C01815=1039.477,-0.924,417.452,169.236,37.751,157.096
C01816=1039.483,-0.675,417.437,169.238,37.752,157.096
C01817=1039.489,-0.426,417.422,169.240,37.752,157.096
C01818=1039.495,-0.176,417.407,169.242,37.753,157.096
C01819=1039.502,0.074,417.392,169.244,37.754,157.096
C01820=1039.508,0.323,417.378,169.246,37.754,157.096
C01821=1039.515,0.572,417.362,169.248,37.754,157.097
C01822=1039.520,0.822,417.347,169.250,37.755,157.097
C01823=1039.526,1.071,417.332,169.253,37.755,157.097
C01824=1039.533,1.321,417.317,169.255,37.756,157.097
C01825=1039.539,1.571,417.302,169.257,37.756,157.097
C01826=1039.545,1.820,417.287,169.259,37.757,157.097
C01827=1039.551,2.069,417.272,169.262,37.758,157.097
C01828=1039.558,2.319,417.257,169.264,37.758,157.098
C01829=1039.564,2.568,417.242,169.266,37.759,157.098
C01830=1039.571,2.817,417.227,169.268,37.759,157.098
C01831=1039.577,3.067,417.212,169.270,37.760,157.098
C01832=1039.583,3.317,417.197,169.272,37.760,157.098
C01833=1039.589,3.566,417.182,169.275,37.761,157.098
C01834=1039.596,3.815,417.167,169.277,37.762,157.098
C01835=1039.602,4.065,417.152,169.279,37.762,157.099
C01836=1039.609,4.314,417.137,169.281,37.763,157.099
C01837=1039.615,4.564,417.122,169.283,37.763,157.099
C01838=1039.621,4.813,417.107,169.285,37.763,157.099
C01839=1039.627,5.063,417.091,169.287,37.764,157.099
C01840=1039.634,5.313,417.076,169.289,37.764,157.099
C01841=1039.640,5.561,417.061,169.291,37.765,157.099
C01842=1039.646,5.811,417.046,169.293,37.766,157.099
C01843=1039.652,6.061,417.031,169.296,37.766,157.099
C01844=1039.659,6.310,417.016,169.298,37.767,157.100
C01845=1039.665,6.559,417.001,169.300,37.767,157.100
C01846=1039.672,6.809,416.986,169.302,37.768,157.100
C01847=1039.678,7.059,416.971,169.304,37.768,157.100
C01848=1039.685,7.308,416.956,169.306,37.769,157.100
C01849=1039.691,7.557,416.940,169.308,37.770,157.100
C01850=1039.698,7.807,416.925,169.310,37.770,157.100
C01851=1039.703,8.057,416.910,169.312,37.770,157.100
C01852=1039.710,8.306,416.894,169.314,37.771,157.101
C01853=1039.716,8.556,416.879,169.316,37.771,157.101
C01854=1039.723,8.805,416.864,169.319,37.772,157.101
C01855=1039.729,9.054,416.849,169.321,37.772,157.101
C01856=1039.735,9.303,416.834,169.322,37.773,157.101
C01857=1039.742,9.553,416.819,169.324,37.774,157.101
C01858=1039.748,9.802,416.803,169.326,37.774,157.101
C01859=1039.755,10.052,416.788,169.328,37.775,157.102
C01860=1039.761,10.301,416.773,169.330,37.775,157.102
C01861=1039.767,10.551,416.757,169.332,37.776,157.102
C01862=1039.773,10.800,416.742,169.334,37.776,157.102
C01863=1039.780,11.049,416.726,169.336,37.777,157.102
C01864=1039.786,11.299,416.711,169.338,37.777,157.102
C01865=1039.793,11.549,416.697,169.341,37.778,157.102
C01866=1039.800,11.798,416.681,169.343,37.778,157.102
C01867=1039.806,12.047,416.666,169.345,37.779,157.102
C01868=1039.813,12.333,416.648,169.348,37.779,157.103
C01869=1039.821,12.618,416.631,169.350,37.780,157.103
C01870=1039.827,12.904,416.613,169.352,37.780,157.103
C01871=1039.835,13.189,416.595,169.354,37.781,157.103
C01872=1039.842,13.438,416.580,169.356,37.782,157.103
C01873=1039.848,13.688,416.565,169.358,37.782,157.103
C01874=1039.855,13.938,416.549,169.361,37.783,157.103
C01875=1039.862,14.187,416.534,169.363,37.783,157.104
C01876=1039.868,14.437,416.517,169.365,37.784,157.104
C01877=1039.874,14.686,416.503,169.367,37.784,157.104
C01878=1039.881,14.935,416.487,169.369,37.785,157.104
C01879=1039.886,15.185,416.471,169.371,37.786,157.104
C01880=1039.893,15.434,416.456,169.373,37.786,157.104
C01881=1039.900,15.683,416.440,169.375,37.787,157.104
C01882=1039.905,15.933,416.424,169.377,37.787,157.105
C01883=1039.912,16.182,416.409,169.379,37.788,157.105
C01884=1039.918,16.432,416.393,169.382,37.788,157.105
C01885=1039.924,16.681,416.378,169.384,37.789,157.105
C01886=1039.931,16.930,416.362,169.386,37.790,157.105
C01887=1039.937,17.180,416.346,169.388,37.791,157.105
C01888=1039.944,17.429,416.331,169.390,37.791,157.105
C01889=1039.949,17.679,416.314,169.392,37.792,157.106
C01890=1039.956,17.928,416.300,169.393,37.793,157.106
C01891=1039.963,18.177,416.284,169.395,37.793,157.106
C01892=1039.968,18.427,416.268,169.397,37.794,157.106
C01893=1039.975,18.677,416.252,169.400,37.794,157.106
C01894=1039.982,18.926,416.237,169.402,37.795,157.106
C01895=1039.988,19.176,416.220,169.404,37.795,157.106
C01896=1039.994,19.425,416.205,169.406,37.796,157.107
C01897=1040.000,19.675,416.189,169.408,37.797,157.107
C01898=1040.007,19.924,416.174,169.410,37.797,157.107
C01899=1040.013,20.174,416.158,169.412,37.798,157.107
C01900=1040.019,20.423,416.142,169.414,37.798,157.107
C01901=1040.025,20.672,416.126,169.416,37.799,157.107
C01902=1040.032,20.921,416.110,169.419,37.799,157.107
C01903=1040.039,21.171,416.094,169.420,37.800,157.107
C01904=1040.045,21.421,416.079,169.422,37.801,157.108
C01905=1040.051,21.670,416.063,169.424,37.802,157.108
C01906=1040.058,21.919,416.047,169.426,37.802,157.108
C01907=1040.064,22.168,416.031,169.428,37.803,157.108
C01908=1040.070,22.417,416.015,169.430,37.804,157.108
C01909=1040.076,22.667,415.999,169.432,37.804,157.108
C01910=1040.083,22.917,415.983,169.434,37.805,157.109
C01911=1040.089,23.167,415.967,169.437,37.805,157.109
C01912=1040.095,23.416,415.951,169.439,37.806,157.109
C01913=1040.102,23.665,415.935,169.441,37.806,157.109
C01914=1040.108,23.914,415.919,169.442,37.808,157.109
C01915=1040.114,24.164,415.904,169.444,37.808,157.109
C01916=1040.120,24.413,415.888,169.446,37.809,157.109
C01917=1040.127,24.663,415.872,169.448,37.809,157.110
C01918=1040.133,24.912,415.855,169.450,37.810,157.110
C01919=1040.140,25.161,415.840,169.452,37.811,157.110
C01920=1040.146,25.411,415.824,169.455,37.811,157.110
C01921=1040.152,25.660,415.807,169.457,37.812,157.110
C01922=1040.159,25.910,415.791,169.459,37.812,157.110
C01923=1040.165,26.159,415.775,169.461,37.813,157.110
C01924=1040.172,26.408,415.759,169.463,37.813,157.111
C01925=1040.178,26.658,415.743,169.464,37.814,157.111
C01926=1040.185,26.907,415.727,169.466,37.815,157.111
C01927=1040.191,27.157,415.711,169.468,37.816,157.111
C01928=1040.197,27.407,415.695,169.470,37.816,157.111
C01929=1040.203,27.656,415.680,169.473,37.817,157.111
C01930=1040.209,27.905,415.663,169.475,37.817,157.111
C01931=1040.216,28.155,415.647,169.477,37.818,157.112
C01932=1040.223,28.441,415.628,169.479,37.819,157.112
C01933=1040.231,28.728,415.609,169.481,37.820,157.112
C01934=1040.238,29.014,415.592,169.483,37.820,157.112
C01935=1040.244,29.301,415.572,169.485,37.821,157.112
C01936=1040.252,29.551,415.556,169.488,37.822,157.113
C01937=1040.258,29.800,415.540,169.490,37.823,157.113
C01938=1040.264,30.049,415.524,169.492,37.823,157.113
C01939=1040.270,30.299,415.508,169.494,37.824,157.113
C01940=1040.276,30.548,415.490,169.496,37.824,157.113
C01941=1040.283,30.797,415.475,169.498,37.826,157.113
C01942=1040.289,31.047,415.458,169.500,37.826,157.113
C01943=1040.295,31.296,415.442,169.501,37.827,157.114
C01944=1040.302,31.546,415.425,169.503,37.827,157.114
C01945=1040.308,31.795,415.410,169.506,37.828,157.114
C01946=1040.314,32.044,415.393,169.508,37.829,157.114
C01947=1040.321,32.293,415.376,169.510,37.830,157.114
C01948=1040.327,32.543,415.360,169.512,37.830,157.114
C01949=1040.333,32.793,415.344,169.514,37.831,157.115
C01950=1040.340,33.042,415.328,169.515,37.832,157.115
C01951=1040.346,33.292,415.311,169.517,37.832,157.115
C01952=1040.352,33.541,415.295,169.519,37.833,157.115
C01953=1040.358,33.790,415.278,169.522,37.834,157.115
C01954=1040.365,34.040,415.261,169.524,37.834,157.115
C01955=1040.372,34.289,415.246,169.526,37.835,157.115
C01956=1040.378,34.538,415.230,169.528,37.836,157.116
C01957=1040.384,34.788,415.213,169.530,37.836,157.116
C01958=1040.390,35.037,415.196,169.531,37.837,157.116
C01959=1040.396,35.286,415.180,169.533,37.838,157.116
C01960=1040.403,35.536,415.163,169.535,37.839,157.116
C01961=1040.410,35.785,415.147,169.537,37.839,157.116
C01962=1040.416,36.034,415.130,169.540,37.840,157.117
C01963=1040.422,36.284,415.114,169.542,37.840,157.117
C01964=1040.428,36.533,415.098,169.544,37.841,157.117
C01965=1040.435,36.782,415.081,169.546,37.841,157.117
C01966=1040.442,37.032,415.065,169.547,37.843,157.117
C01967=1040.448,37.281,415.048,169.549,37.843,157.117
C01968=1040.454,37.531,415.032,169.551,37.844,157.117
C01969=1040.461,37.780,415.015,169.553,37.844,157.118
C01970=1040.467,38.029,414.998,169.556,37.845,157.118
C01971=1040.473,38.278,414.981,169.558,37.846,157.118
C01972=1040.479,38.528,414.965,169.559,37.847,157.118
C01973=1040.485,38.778,414.949,169.561,37.847,157.118
C01974=1040.492,39.027,414.931,169.563,37.848,157.119
C01975=1040.498,39.276,414.915,169.565,37.849,157.119
C01976=1040.505,39.525,414.898,169.567,37.850,157.119
C01977=1040.510,39.775,414.881,169.569,37.850,157.119
C01978=1040.516,40.025,414.865,169.571,37.851,157.119
C01979=1040.523,40.273,414.848,169.573,37.852,157.119
C01980=1040.529,40.524,414.831,169.575,37.853,157.119
C01981=1040.535,40.772,414.814,169.577,37.853,157.120
C01982=1040.542,41.022,414.797,169.579,37.854,157.120
C01983=1040.548,41.271,414.780,169.581,37.855,157.120
C01984=1040.554,41.520,414.764,169.582,37.855,157.120
C01985=1040.561,41.770,414.747,169.584,37.856,157.120
C01986=1040.567,42.019,414.731,169.587,37.857,157.121
C01987=1040.574,42.269,414.713,169.589,37.858,157.121
C01988=1040.580,42.518,414.697,169.591,37.858,157.121
C01989=1040.586,42.767,414.680,169.593,37.859,157.121
C01990=1040.593,43.017,414.663,169.594,37.860,157.121
C01991=1040.599,43.265,414.646,169.596,37.861,157.121
C01992=1040.605,43.516,414.629,169.598,37.861,157.121
C01993=1040.611,43.765,414.612,169.601,37.862,157.122
C01994=1040.617,44.015,414.596,169.603,37.863,157.122
C01995=1040.624,44.263,414.579,169.605,37.864,157.122
C01996=1040.630,44.550,414.559,169.607,37.865,157.122
C01997=1040.638,44.837,414.539,169.609,37.865,157.122
C01998=1040.645,45.123,414.520,169.611,37.867,157.123
C01999=1040.652,45.410,414.500,169.614,37.868,157.123
C02000=1040.658,45.659,414.483,169.616,37.868,157.123
C02001=1040.664,45.908,414.466,169.617,37.869,157.123
C02002=1040.670,46.158,414.449,169.619,37.870,157.123
C02003=1040.676,46.407,414.432,169.621,37.871,157.124
C02004=1040.682,46.657,414.414,169.623,37.871,157.124
C02005=1040.688,46.906,414.398,169.625,37.873,157.124
C02006=1040.695,47.155,414.381,169.626,37.873,157.124
C02007=1040.701,47.404,414.363,169.629,37.874,157.124
C02008=1040.707,47.654,414.347,169.631,37.875,157.125
C02009=1040.714,47.903,414.329,169.633,37.875,157.125
C02010=1040.720,48.152,414.312,169.635,37.876,157.125
C02011=1040.726,48.402,414.294,169.636,37.877,157.125
C02012=1040.732,48.651,414.278,169.638,37.878,157.125
C02013=1040.739,48.900,414.261,169.640,37.879,157.125
C02014=1040.744,49.150,414.243,169.643,37.880,157.126
C02015=1040.751,49.399,414.226,169.645,37.880,157.126
C02016=1040.757,49.648,414.210,169.646,37.881,157.126
C02017=1040.763,49.898,414.192,169.648,37.882,157.126
C02018=1040.770,50.147,414.175,169.650,37.883,157.126
C02019=1040.776,50.396,414.157,169.652,37.884,157.126
C02020=1040.782,50.645,414.140,169.654,37.884,157.127
C02021=1040.788,50.895,414.123,169.656,37.885,157.127
C02022=1040.795,51.144,414.106,169.658,37.886,157.127
C02023=1040.801,51.394,414.088,169.660,37.887,157.127
C02024=1040.809,51.733,414.065,169.663,37.888,157.127
C02025=1040.818,52.073,414.041,169.665,37.888,157.128
C02026=1040.827,52.412,414.018,169.667,37.890,157.128
C02027=1040.835,52.751,413.995,169.671,37.891,157.128
C02028=1040.841,53.001,413.977,169.673,37.891,157.128
C02029=1040.847,53.250,413.960,169.675,37.893,157.128
C02030=1040.854,53.500,413.943,169.676,37.893,157.129
C02031=1040.860,53.749,413.925,169.678,37.894,157.129
C02032=1040.866,53.998,413.908,169.680,37.895,157.129
C02033=1040.873,54.247,413.891,169.682,37.895,157.129
C02034=1040.879,54.497,413.873,169.685,37.896,157.129
C02035=1040.886,54.746,413.856,169.686,37.897,157.130
C02036=1040.893,54.995,413.839,169.688,37.898,157.130
C02037=1040.898,55.244,413.821,169.690,37.898,157.130
C02038=1040.905,55.494,413.804,169.692,37.899,157.130
C02039=1040.910,55.743,413.787,169.694,37.900,157.130
C02040=1040.917,55.993,413.769,169.695,37.901,157.130
C02041=1040.924,56.242,413.752,169.697,37.901,157.130
C02042=1040.929,56.491,413.735,169.700,37.903,157.131
C02043=1040.936,56.741,413.717,169.702,37.903,157.131
C02044=1040.943,56.990,413.700,169.704,37.904,157.131
C02045=1040.949,57.239,413.682,169.705,37.904,157.131
C02046=1040.955,57.489,413.665,169.707,37.905,157.131
C02047=1040.961,57.738,413.647,169.709,37.906,157.132
C02048=1040.968,57.987,413.630,169.711,37.907,157.132
C02049=1040.975,58.237,413.613,169.714,37.908,157.132
C02050=1040.980,58.486,413.595,169.715,37.908,157.132
C02051=1040.987,58.735,413.578,169.717,37.909,157.132
C02052=1040.993,58.985,413.560,169.719,37.910,157.132
C02053=1041.000,59.234,413.543,169.721,37.911,157.133
C02054=1041.006,59.483,413.526,169.723,37.911,157.133
C02055=1041.013,59.732,413.507,169.725,37.912,157.133
C02056=1041.019,59.955,413.492,169.726,37.912,157.133
C02057=1041.024,60.178,413.476,169.729,37.913,157.133
C02058=1041.030,60.401,413.461,169.730,37.914,157.133
C02059=1041.036,60.623,413.445,169.732,37.915,157.134
C02060=1041.041,60.845,413.429,169.734,37.915,157.134
C02061=1041.047,61.068,413.413,169.735,37.916,157.134
C02062=1041.053,61.292,413.398,169.737,37.917,157.134
C02063=1041.058,61.514,413.382,169.739,37.917,157.134
C02064=1041.065,61.763,413.365,169.740,37.918,157.134
C02065=1041.071,62.013,413.347,169.743,37.919,157.134
C02066=1041.078,62.262,413.329,169.745,37.919,157.135
C02067=1041.084,62.511,413.312,169.747,37.920,157.135
C02068=1041.091,62.760,413.294,169.749,37.921,157.135
C02069=1041.097,63.010,413.276,169.750,37.922,157.135
C02070=1041.104,63.259,413.259,169.752,37.922,157.135
C02071=1041.110,63.508,413.242,169.754,37.923,157.135
C02072=1041.116,63.757,413.223,169.756,37.923,157.136
C02073=1041.123,64.007,413.206,169.759,37.925,157.136
C02074=1041.129,64.257,413.188,169.760,37.925,157.136
C02075=1041.135,64.506,413.171,169.762,37.926,157.136
C02076=1041.142,64.755,413.153,169.764,37.927,157.136
C02077=1041.148,65.004,413.135,169.766,37.928,157.136
C02078=1041.154,65.254,413.117,169.768,37.929,157.137
C02079=1041.160,65.503,413.100,169.769,37.929,157.137
C02080=1041.167,65.752,413.081,169.772,37.930,157.137
C02081=1041.173,66.001,413.063,169.774,37.931,157.137
C02082=1041.179,66.251,413.045,169.776,37.932,157.137
C02083=1041.185,66.500,413.028,169.778,37.933,157.138
C02084=1041.192,66.749,413.010,169.779,37.933,157.138
C02085=1041.198,66.999,412.992,169.781,37.934,157.138
C02086=1041.205,67.248,412.974,169.783,37.935,157.138
C02087=1041.211,67.497,412.956,169.786,37.936,157.138
C02088=1041.217,67.746,412.938,169.787,37.936,157.138
C02089=1041.223,67.995,412.919,169.789,37.938,157.139
C02090=1041.230,68.245,412.902,169.791,37.938,157.139
C02091=1041.236,68.495,412.884,169.793,37.939,157.139
C02092=1041.242,68.743,412.866,169.795,37.940,157.139
C02093=1041.248,68.993,412.848,169.796,37.940,157.139
C02094=1041.255,69.242,412.831,169.799,37.942,157.140
C02095=1041.261,69.491,412.812,169.801,37.942,157.140
C02096=1041.267,69.740,412.794,169.803,37.943,157.140
C02097=1041.273,69.990,412.776,169.804,37.944,157.140
C02098=1041.279,70.239,412.758,169.806,37.945,157.140
C02099=1041.286,70.488,412.739,169.808,37.946,157.141
C02100=1041.293,70.738,412.722,169.810,37.946,157.141
C02101=1041.299,70.986,412.703,169.813,37.948,157.141
C02102=1041.305,71.236,412.686,169.814,37.948,157.141
C02103=1041.311,71.485,412.667,169.816,37.949,157.141
C02104=1041.317,71.735,412.649,169.818,37.950,157.142
C02105=1041.324,71.984,412.630,169.820,37.951,157.142
C02106=1041.329,72.233,412.613,169.821,37.952,157.142
C02107=1041.336,72.482,412.594,169.824,37.953,157.142
C02108=1041.342,72.732,412.576,169.826,37.953,157.142
C02109=1041.349,72.981,412.558,169.828,37.954,157.142
C02110=1041.355,73.230,412.540,169.830,37.955,157.143
C02111=1041.361,73.480,412.522,169.831,37.956,157.143
C02112=1041.367,73.729,412.504,169.833,37.957,157.143
C02113=1041.373,73.978,412.485,169.835,37.958,157.143
C02114=1041.380,74.227,412.467,169.838,37.959,157.144
C02115=1041.386,74.477,412.449,169.839,37.959,157.144
C02116=1041.392,74.726,412.430,169.841,37.960,157.144
C02117=1041.398,74.975,412.412,169.843,37.961,157.144
C02118=1041.405,75.225,412.394,169.845,37.962,157.144
C02119=1041.411,75.473,412.375,169.847,37.963,157.144
C02120=1041.417,75.723,412.357,169.849,37.963,157.145
C02121=1041.423,75.972,412.339,169.851,37.965,157.145
C02122=1041.430,76.221,412.321,169.853,37.965,157.145
C02123=1041.437,76.470,412.303,169.855,37.966,157.145
C02124=1041.444,76.757,412.281,169.857,37.967,157.145
C02125=1041.451,77.042,412.260,169.859,37.968,157.146
C02126=1041.458,77.329,412.239,169.861,37.969,157.146
C02127=1041.465,77.615,412.218,169.864,37.970,157.146
C02128=1041.471,77.864,412.199,169.866,37.970,157.146
C02129=1041.477,78.113,412.181,169.867,37.972,157.146
C02130=1041.483,78.363,412.163,169.869,37.972,157.147
C02131=1041.490,78.612,412.144,169.871,37.973,157.147
C02132=1041.496,78.861,412.126,169.873,37.974,157.147
C02133=1041.503,79.110,412.107,169.875,37.975,157.147
C02134=1041.509,79.360,412.089,169.877,37.976,157.148
C02135=1041.514,79.609,412.070,169.879,37.977,157.148
C02136=1041.521,79.858,412.051,169.881,37.978,157.148
C02137=1041.527,80.107,412.033,169.882,37.979,157.148
C02138=1041.533,80.356,412.014,169.884,37.980,157.148
C02139=1041.539,80.605,411.996,169.887,37.980,157.148
C02140=1041.545,80.855,411.977,169.889,37.982,157.149
C02141=1041.551,81.104,411.958,169.891,37.982,157.149
C02142=1041.558,81.353,411.940,169.892,37.983,157.149
C02143=1041.564,81.602,411.921,169.894,37.984,157.149
C02144=1041.571,81.851,411.902,169.896,37.985,157.150
C02145=1041.576,82.101,411.883,169.899,37.986,157.150
C02146=1041.582,82.351,411.865,169.900,37.987,157.150
C02147=1041.589,82.600,411.847,169.902,37.987,157.150
C02148=1041.595,82.849,411.828,169.904,37.989,157.150
C02149=1041.602,83.098,411.809,169.906,37.989,157.150
C02150=1041.607,83.347,411.790,169.907,37.990,157.151
C02151=1041.614,83.597,411.771,169.909,37.991,157.151
C02152=1041.620,83.846,411.753,169.912,37.992,157.151
C02153=1041.627,84.095,411.734,169.914,37.993,157.151
C02154=1041.633,84.344,411.716,169.916,37.994,157.152
C02155=1041.639,84.593,411.696,169.917,37.994,157.152
C02156=1041.645,84.842,411.678,169.919,37.996,157.152
C02157=1041.652,85.092,411.659,169.921,37.996,157.152
C02158=1041.658,85.341,411.641,169.924,37.997,157.152
C02159=1041.664,85.590,411.622,169.925,37.998,157.152
C02160=1041.670,85.840,411.603,169.927,37.999,157.153
C02161=1041.676,86.089,411.585,169.929,38.000,157.153
C02162=1041.683,86.338,411.566,169.931,38.001,157.153
C02163=1041.689,86.587,411.547,169.933,38.001,157.153
C02164=1041.695,86.837,411.528,169.935,38.003,157.153
C02165=1041.701,87.086,411.509,169.937,38.003,157.154
C02166=1041.708,87.335,411.491,169.939,38.004,157.154
C02167=1041.714,87.584,411.472,169.941,38.005,157.154
C02168=1041.720,87.833,411.453,169.942,38.006,157.154
C02169=1041.726,88.083,411.434,169.944,38.007,157.154
C02170=1041.733,88.331,411.415,169.947,38.008,157.155
C02171=1041.739,88.580,411.396,169.949,38.009,157.155
C02172=1041.746,88.829,411.377,169.951,38.010,157.155
C02173=1041.751,89.079,411.358,169.952,38.010,157.155
C02174=1041.758,89.328,411.340,169.954,38.011,157.155
C02175=1041.764,89.577,411.321,169.956,38.012,157.156
C02176=1041.771,89.826,411.302,169.958,38.013,157.156
C02177=1041.777,90.076,411.283,169.961,38.014,157.156
C02178=1041.783,90.325,411.264,169.962,38.014,157.156
C02179=1041.789,90.575,411.245,169.964,38.016,157.156
C02180=1041.796,90.823,411.225,169.966,38.017,157.157
C02181=1041.802,91.073,411.206,169.968,38.017,157.157
C02182=1041.808,91.322,411.188,169.969,38.019,157.157
C02183=1041.814,91.571,411.168,169.972,38.019,157.157
C02184=1041.820,91.820,411.150,169.974,38.020,157.157
C02185=1041.826,92.069,411.130,169.976,38.021,157.158
C02186=1041.833,92.318,411.111,169.977,38.022,157.158
C02187=1041.838,92.568,411.092,169.979,38.023,157.158
C02188=1041.845,92.854,411.070,169.982,38.024,157.158
C02189=1041.853,93.140,411.048,169.984,38.025,157.159
C02190=1041.860,93.426,411.026,169.986,38.026,157.159
C02191=1041.867,93.712,411.004,169.988,38.027,157.159
C02192=1041.873,93.961,410.985,169.990,38.028,157.159
C02193=1041.879,94.210,410.966,169.992,38.029,157.159
C02194=1041.885,94.459,410.946,169.995,38.030,157.160
C02195=1041.892,94.708,410.927,169.996,38.031,157.160
C02196=1041.898,94.958,410.908,169.998,38.032,157.160
C02197=1041.904,95.206,410.889,170.000,38.033,157.160
C02198=1041.911,95.456,410.869,170.002,38.034,157.161
C02199=1041.917,95.706,410.850,170.004,38.035,157.161
C02200=1041.923,95.955,410.831,170.006,38.036,157.161
C02201=1041.929,96.204,410.811,170.008,38.037,157.161
C02202=1041.935,96.453,410.793,170.010,38.037,157.161
C02203=1041.941,96.702,410.773,170.012,38.038,157.162
C02204=1041.948,96.951,410.754,170.014,38.039,157.162
C02205=1041.954,97.201,410.734,170.015,38.040,157.162
C02206=1041.961,97.449,410.715,170.018,38.041,157.162
C02207=1041.966,97.699,410.696,170.020,38.042,157.162
C02208=1041.973,97.948,410.677,170.022,38.043,157.163
C02209=1041.979,98.197,410.657,170.024,38.044,157.163
C02210=1041.985,98.446,410.639,170.025,38.045,157.163
C02211=1041.992,98.695,410.618,170.027,38.045,157.163
C02212=1041.997,98.945,410.599,170.030,38.047,157.163
C02213=1042.004,99.194,410.580,170.032,38.047,157.164
C02214=1042.010,99.443,410.560,170.034,38.048,157.164
C02215=1042.016,99.692,410.542,170.035,38.049,157.164
C02216=1042.023,99.941,410.521,170.037,38.050,157.164
C02217=1042.029,100.191,410.503,170.039,38.051,157.165
C02218=1042.035,100.439,410.483,170.042,38.052,157.165
C02219=1042.041,100.689,410.464,170.044,38.053,157.165
C02220=1042.048,100.937,410.444,170.045,38.054,157.165
C02221=1042.054,101.188,410.425,170.047,38.055,157.165
C02222=1042.060,101.436,410.405,170.049,38.056,157.166
C02223=1042.066,101.686,410.385,170.051,38.056,157.166
C02224=1042.072,101.935,410.365,170.053,38.058,157.166
C02225=1042.078,102.183,410.345,170.055,38.059,157.166
C02226=1042.085,102.433,410.326,170.057,38.059,157.166
C02227=1042.091,102.682,410.306,170.059,38.061,157.167
C02228=1042.096,102.931,410.287,170.061,38.062,157.167
C02229=1042.102,103.180,410.267,170.062,38.062,157.167
C02230=1042.108,103.429,410.247,170.065,38.064,157.167
C02231=1042.115,103.679,410.228,170.067,38.065,157.168
C02232=1042.121,103.928,410.208,170.069,38.065,157.168
C02233=1042.127,104.177,410.189,170.070,38.067,157.168
C02234=1042.133,104.426,410.169,170.072,38.068,157.168
C02235=1042.140,104.675,410.149,170.075,38.068,157.168
C02236=1042.146,104.925,410.130,170.077,38.069,157.169
C02237=1042.152,105.173,410.110,170.079,38.071,157.169
C02238=1042.158,105.422,410.090,170.080,38.071,157.169
C02239=1042.164,105.672,410.071,170.082,38.072,157.169
C02240=1042.170,105.921,410.051,170.085,38.074,157.170
C02241=1042.176,106.170,410.031,170.087,38.074,157.170
C02242=1042.183,106.419,410.012,170.089,38.075,157.170
C02243=1042.189,106.669,409.992,170.090,38.076,157.170
C02244=1042.195,106.917,409.972,170.092,38.077,157.170
C02245=1042.201,107.166,409.952,170.094,38.078,157.171
C02246=1042.208,107.416,409.932,170.096,38.079,157.171
C02247=1042.214,107.665,409.912,170.099,38.080,157.171
C02248=1042.220,107.914,409.893,170.100,38.081,157.171
C02249=1042.227,108.163,409.873,170.102,38.082,157.172
C02250=1042.233,108.413,409.853,170.104,38.083,157.172
C02251=1042.239,108.661,409.833,170.106,38.084,157.172
C02252=1042.245,108.947,409.810,170.109,38.085,157.172
C02253=1042.253,109.234,409.788,170.111,38.086,157.172
C02254=1042.260,109.520,409.765,170.113,38.087,157.173
C02255=1042.267,109.806,409.742,170.115,38.088,157.173
C02256=1042.273,110.054,409.722,170.117,38.089,157.173
C02257=1042.280,110.304,409.702,170.120,38.090,157.173
C02258=1042.286,110.553,409.682,170.122,38.091,157.174
C02259=1042.292,110.802,409.662,170.124,38.092,157.174
C02260=1042.298,111.052,409.643,170.125,38.093,157.174
C02261=1042.304,111.300,409.623,170.127,38.094,157.174
C02262=1042.310,111.549,409.603,170.130,38.095,157.175
C02263=1042.317,111.799,409.582,170.132,38.096,157.175
C02264=1042.323,112.048,409.562,170.134,38.097,157.175
C02265=1042.329,112.296,409.542,170.135,38.098,157.175
C02266=1042.336,112.546,409.522,170.137,38.099,157.175
C02267=1042.342,112.795,409.502,170.139,38.100,157.176
C02268=1042.348,113.044,409.482,170.142,38.101,157.176
C02269=1042.354,113.293,409.462,170.144,38.101,157.176
C02270=1042.360,113.542,409.442,170.146,38.103,157.176
C02271=1042.367,113.791,409.422,170.147,38.104,157.177
C02272=1042.373,114.040,409.402,170.149,38.105,157.177
C02273=1042.378,114.289,409.381,170.151,38.106,157.177
C02274=1042.385,114.539,409.361,170.154,38.107,157.177
C02275=1042.391,114.788,409.341,170.156,38.108,157.178
C02276=1042.397,115.037,409.321,170.157,38.109,157.178
C02277=1042.402,115.286,409.300,170.159,38.110,157.178
C02278=1042.408,115.535,409.280,170.162,38.111,157.178
C02279=1042.414,115.784,409.260,170.164,38.112,157.178
C02280=1042.420,116.034,409.239,170.166,38.113,157.179
C02281=1042.426,116.283,409.219,170.167,38.114,157.179
C02282=1042.433,116.532,409.199,170.169,38.116,157.179
C02283=1042.439,116.780,409.178,170.172,38.117,157.180
C02284=1042.444,117.029,409.158,170.174,38.117,157.180
C02285=1042.451,117.279,409.137,170.176,38.118,157.180
C02286=1042.457,117.528,409.117,170.177,38.120,157.180
C02287=1042.462,117.777,409.097,170.179,38.121,157.180
C02288=1042.469,118.026,409.076,170.181,38.122,157.181
C02289=1042.475,118.275,409.056,170.184,38.123,157.181
C02290=1042.481,118.525,409.036,170.186,38.124,157.181
C02291=1042.487,118.773,409.015,170.188,38.125,157.181
C02292=1042.494,119.023,408.995,170.189,38.126,157.182
C02293=1042.500,119.272,408.975,170.191,38.127,157.182
C02294=1042.505,119.521,408.954,170.194,38.128,157.182
C02295=1042.511,119.770,408.934,170.196,38.129,157.182
C02296=1042.518,120.018,408.913,170.198,38.130,157.183
C02297=1042.524,120.268,408.893,170.199,38.131,157.183
C02298=1042.530,120.517,408.872,170.201,38.133,157.183
C02299=1042.536,120.767,408.852,170.204,38.133,157.183
C02300=1042.542,121.015,408.831,170.206,38.134,157.184
C02301=1042.548,121.265,408.810,170.208,38.135,157.184
C02302=1042.554,121.513,408.790,170.210,38.137,157.184
C02303=1042.561,121.763,408.770,170.212,38.137,157.184
C02304=1042.566,122.011,408.749,170.214,38.138,157.184
C02305=1042.572,122.260,408.729,170.216,38.140,157.185
C02306=1042.579,122.510,408.708,170.218,38.141,157.185
C02307=1042.584,122.759,408.688,170.220,38.142,157.185
C02308=1042.591,123.008,408.667,170.222,38.142,157.185
C02309=1042.597,123.257,408.647,170.225,38.144,157.186
C02310=1042.603,123.506,408.626,170.226,38.145,157.186
C02311=1042.610,123.755,408.605,170.228,38.146,157.186
C02312=1042.616,124.004,408.585,170.230,38.147,157.186
C02313=1042.622,124.254,408.564,170.232,38.148,157.187
C02314=1042.628,124.502,408.543,170.235,38.149,157.187
C02315=1042.635,124.752,408.523,170.237,38.150,157.187
C02316=1042.642,125.037,408.499,170.239,38.151,157.187
C02317=1042.649,125.322,408.476,170.241,38.152,157.188
C02318=1042.656,125.609,408.452,170.243,38.154,157.188
C02319=1042.662,125.895,408.428,170.246,38.155,157.188
C02320=1042.669,126.144,408.407,170.248,38.155,157.188
C02321=1042.675,126.393,408.387,170.250,38.156,157.189
C02322=1042.681,126.642,408.366,170.252,38.158,157.189
C02323=1042.688,126.891,408.345,170.254,38.159,157.189
C02324=1042.694,127.140,408.325,170.256,38.159,157.189
C02325=1042.700,127.389,408.304,170.259,38.160,157.190
C02326=1042.706,127.638,408.284,170.261,38.162,157.190
C02327=1042.713,127.887,408.263,170.262,38.163,157.190
C02328=1042.719,128.137,408.242,170.264,38.163,157.190
C02329=1042.725,128.385,408.221,170.266,38.164,157.191
C02330=1042.732,128.635,408.201,170.269,38.166,157.191
C02331=1042.737,128.883,408.179,170.271,38.167,157.191
C02332=1042.744,129.133,408.159,170.273,38.167,157.191
C02333=1042.751,129.381,408.138,170.275,38.169,157.191
C02334=1042.756,129.631,408.117,170.277,38.170,157.192
C02335=1042.763,129.879,408.096,170.280,38.171,157.192
C02336=1042.769,130.129,408.076,170.281,38.171,157.192
C02337=1042.775,130.377,408.055,170.283,38.173,157.192
C02338=1042.782,130.627,408.035,170.285,38.174,157.193
C02339=1042.788,130.876,408.013,170.287,38.175,157.193
C02340=1042.794,131.125,407.993,170.290,38.175,157.193
C02341=1042.800,131.374,407.971,170.292,38.177,157.193
C02342=1042.807,131.623,407.950,170.294,38.178,157.194
C02343=1042.812,131.872,407.930,170.296,38.179,157.194
C02344=1042.818,132.121,407.908,170.298,38.180,157.194
C02345=1042.825,132.370,407.887,170.301,38.181,157.194
C02346=1042.830,132.619,407.866,170.302,38.183,157.195
C02347=1042.837,132.869,407.845,170.304,38.184,157.195
C02348=1042.843,133.117,407.824,170.306,38.185,157.195
C02349=1042.849,133.367,407.803,170.308,38.185,157.195
C02350=1042.855,133.616,407.782,170.311,38.187,157.196
C02351=1042.861,133.864,407.761,170.313,38.188,157.196
C02352=1042.867,134.114,407.740,170.315,38.189,157.196
C02353=1042.873,134.363,407.718,170.317,38.190,157.196
C02354=1042.880,134.611,407.698,170.320,38.191,157.197
C02355=1042.886,134.861,407.676,170.321,38.192,157.197
C02356=1042.892,135.110,407.655,170.323,38.194,157.197
C02357=1042.898,135.359,407.634,170.325,38.195,157.198
C02358=1042.904,135.608,407.613,170.327,38.195,157.198
C02359=1042.910,135.857,407.591,170.330,38.196,157.198
C02360=1042.917,136.105,407.571,170.332,38.198,157.198
C02361=1042.922,136.355,407.550,170.334,38.199,157.198
C02362=1042.929,136.604,407.528,170.336,38.200,157.199
C02363=1042.935,136.852,407.507,170.338,38.201,157.199
C02364=1042.941,137.102,407.486,170.341,38.202,157.199
C02365=1042.947,137.351,407.464,170.343,38.203,157.200
C02366=1042.953,137.600,407.442,170.344,38.205,157.200
C02367=1042.959,137.849,407.422,170.346,38.206,157.200
C02368=1042.966,138.098,407.401,170.348,38.206,157.200
C02369=1042.972,138.347,407.379,170.351,38.207,157.200
C02370=1042.978,138.596,407.358,170.353,38.209,157.201
C02371=1042.983,138.845,407.336,170.355,38.210,157.201
C02372=1042.990,139.094,407.315,170.357,38.211,157.201
C02373=1042.996,139.343,407.294,170.360,38.212,157.202
C02374=1043.003,139.592,407.272,170.362,38.213,157.202
C02375=1043.008,139.841,407.251,170.364,38.214,157.202
C02376=1043.014,140.090,407.229,170.366,38.216,157.202
C02377=1043.021,140.339,407.207,170.368,38.217,157.203
C02378=1043.026,140.588,407.186,170.371,38.218,157.203
C02379=1043.032,140.837,407.164,170.372,38.219,157.203
C02380=1043.040,141.123,407.140,170.375,38.220,157.203
C02381=1043.046,141.408,407.115,170.377,38.222,157.204
C02382=1043.053,141.694,407.091,170.380,38.223,157.204
C02383=1043.061,141.979,407.067,170.382,38.224,157.204
C02384=1043.067,142.228,407.045,170.384,38.225,157.205
C02385=1043.073,142.478,407.023,170.386,38.227,157.205
C02386=1043.079,142.727,407.002,170.389,38.228,157.205
C02387=1043.085,142.975,406.980,170.391,38.229,157.205
C02388=1043.091,143.225,406.959,170.393,38.230,157.206
C02389=1043.097,143.474,406.937,170.395,38.231,157.206
C02390=1043.103,143.723,406.915,170.397,38.232,157.206
C02391=1043.110,143.972,406.893,170.400,38.234,157.207
C02392=1043.115,144.220,406.872,170.402,38.235,157.207
C02393=1043.121,144.469,406.850,170.404,38.236,157.207
C02394=1043.127,144.718,406.829,170.406,38.237,157.207
C02395=1043.134,144.968,406.807,170.409,38.238,157.208
C02396=1043.140,145.217,406.785,170.411,38.239,157.208
C02397=1043.146,145.466,406.764,170.413,38.240,157.208
C02398=1043.152,145.715,406.742,170.415,38.242,157.208
C02399=1043.158,145.963,406.720,170.417,38.243,157.209
C02400=1043.165,146.212,406.699,170.420,38.244,157.209
C02401=1043.171,146.461,406.677,170.422,38.245,157.209
C02402=1043.177,146.710,406.656,170.423,38.246,157.210
C02403=1043.183,146.960,406.634,170.425,38.247,157.210
C02404=1043.190,147.208,406.612,170.428,38.249,157.210
C02405=1043.195,147.457,406.590,170.430,38.250,157.210
C02406=1043.201,147.706,406.568,170.432,38.251,157.211
C02407=1043.207,147.955,406.547,170.434,38.252,157.211
C02408=1043.213,148.204,406.524,170.436,38.253,157.211
C02409=1043.220,148.453,406.503,170.439,38.254,157.211
C02410=1043.226,148.702,406.481,170.441,38.256,157.212
C02411=1043.232,148.951,406.459,170.443,38.257,157.212
C02412=1043.238,149.200,406.437,170.445,38.258,157.212
C02413=1043.243,149.449,406.415,170.448,38.259,157.213
C02414=1043.250,149.698,406.393,170.450,38.261,157.213
C02415=1043.256,149.947,406.371,170.452,38.262,157.213
C02416=1043.262,150.196,406.349,170.454,38.263,157.213
C02417=1043.269,150.445,406.327,170.457,38.264,157.214
C02418=1043.274,150.694,406.305,170.459,38.265,157.214
C02419=1043.280,150.943,406.283,170.461,38.267,157.214
C02420=1043.287,151.192,406.261,170.463,38.268,157.215
C02421=1043.293,151.441,406.239,170.465,38.269,157.215
C02422=1043.299,151.689,406.217,170.468,38.270,157.215
C02423=1043.304,151.939,406.195,170.470,38.271,157.215
C02424=1043.311,152.187,406.173,170.472,38.273,157.216
C02425=1043.317,152.436,406.151,170.474,38.274,157.216
C02426=1043.323,152.686,406.129,170.477,38.275,157.216
C02427=1043.329,152.934,406.107,170.479,38.276,157.217
C02428=1043.335,153.184,406.085,170.481,38.278,157.217
C02429=1043.341,153.432,406.063,170.483,38.279,157.217
C02430=1043.347,153.681,406.041,170.486,38.280,157.217
C02431=1043.354,153.930,406.019,170.488,38.281,157.218
C02432=1043.359,154.180,405.996,170.490,38.282,157.218
C02433=1043.366,154.428,405.974,170.492,38.284,157.218
C02434=1043.372,154.677,405.952,170.495,38.285,157.219
C02435=1043.378,154.926,405.929,170.497,38.286,157.219
C02436=1043.384,155.175,405.907,170.499,38.287,157.219
C02437=1043.390,155.424,405.885,170.501,38.289,157.219
C02438=1043.396,155.673,405.862,170.503,38.290,157.220
C02439=1043.402,155.922,405.841,170.506,38.291,157.220
C02440=1043.409,156.171,405.818,170.508,38.293,157.220
C02441=1043.414,156.420,405.795,170.510,38.294,157.221
C02442=1043.421,156.669,405.774,170.513,38.295,157.221
C02443=1043.427,156.917,405.752,170.515,38.296,157.221
C02444=1043.433,157.203,405.726,170.518,38.298,157.222
C02445=1043.440,157.488,405.700,170.520,38.299,157.222
C02446=1043.447,157.774,405.675,170.523,38.301,157.222
C02447=1043.454,158.058,405.649,170.526,38.302,157.223
C02448=1043.461,158.307,405.627,170.528,38.303,157.223
C02449=1043.466,158.556,405.604,170.530,38.305,157.223
C02450=1043.473,158.805,405.582,170.533,38.306,157.223
C02451=1043.478,159.054,405.560,170.535,38.307,157.224
C02452=1043.485,159.303,405.537,170.537,38.308,157.224
C02453=1043.492,159.552,405.515,170.539,38.309,157.224
C02454=1043.497,159.801,405.492,170.542,38.311,157.225
C02455=1043.504,160.050,405.470,170.544,38.312,157.225
C02456=1043.510,160.299,405.448,170.546,38.313,157.225
C02457=1043.516,160.548,405.425,170.548,38.315,157.226
C02458=1043.522,160.797,405.402,170.551,38.316,157.226
C02459=1043.527,161.046,405.380,170.553,38.317,157.226
C02460=1043.533,161.295,405.357,170.555,38.319,157.226
C02461=1043.539,161.544,405.334,170.557,38.320,157.227
C02462=1043.545,161.793,405.311,170.560,38.322,157.227
C02463=1043.551,162.042,405.288,170.562,38.323,157.228
C02464=1043.556,162.290,405.265,170.564,38.324,157.228
C02465=1043.563,162.539,405.243,170.566,38.326,157.228
C02466=1043.569,162.788,405.220,170.569,38.327,157.228
C02467=1043.574,163.037,405.197,170.571,38.329,157.229
C02468=1043.580,163.286,405.174,170.573,38.330,157.229
C02469=1043.586,163.535,405.151,170.576,38.331,157.229
C02470=1043.592,163.783,405.129,170.578,38.333,157.230
C02471=1043.598,164.032,405.106,170.580,38.334,157.230
C02472=1043.604,164.281,405.083,170.583,38.335,157.230
C02473=1043.609,164.530,405.060,170.586,38.337,157.231
C02474=1043.615,164.779,405.037,170.588,38.338,157.231
C02475=1043.622,165.027,405.015,170.590,38.340,157.231
C02476=1043.628,165.277,404.992,170.593,38.341,157.232
C02477=1043.634,165.526,404.969,170.595,38.342,157.232
C02478=1043.639,165.775,404.946,170.597,38.344,157.232
C02479=1043.645,166.024,404.923,170.599,38.345,157.233
C02480=1043.652,166.272,404.900,170.602,38.346,157.233
C02481=1043.657,166.521,404.877,170.604,38.348,157.233
C02482=1043.663,166.770,404.854,170.606,38.349,157.234
C02483=1043.669,167.019,404.832,170.608,38.351,157.234
C02484=1043.675,167.268,404.809,170.611,38.352,157.234
C02485=1043.681,167.517,404.785,170.613,38.354,157.235
C02486=1043.687,167.766,404.763,170.615,38.355,157.235
C02487=1043.693,168.014,404.739,170.619,38.356,157.235
C02488=1043.699,168.263,404.716,170.621,38.358,157.236
C02489=1043.705,168.512,404.693,170.623,38.359,157.236
C02490=1043.711,168.761,404.670,170.625,38.361,157.236
C02491=1043.718,169.010,404.648,170.628,38.362,157.237
C02492=1043.723,169.259,404.625,170.630,38.363,157.237
C02493=1043.729,169.507,404.601,170.632,38.365,157.237
C02494=1043.735,169.756,404.578,170.634,38.366,157.238
C02495=1043.741,170.005,404.555,170.637,38.368,157.238
C02496=1043.747,170.254,404.532,170.640,38.369,157.238
C02497=1043.753,170.504,404.509,170.642,38.371,157.239
C02498=1043.760,170.752,404.486,170.645,38.372,157.239
C02499=1043.765,171.001,404.463,170.647,38.373,157.239
C02500=1043.771,171.250,404.440,170.649,38.375,157.240
C02501=1043.777,171.499,404.417,170.651,38.376,157.240
C02502=1043.784,171.747,404.393,170.654,38.378,157.240
C02503=1043.789,171.996,404.370,170.656,38.379,157.241
C02504=1043.796,172.245,404.348,170.659,38.381,157.241
C02505=1043.802,172.494,404.324,170.662,38.382,157.241
C02506=1043.808,172.743,404.301,170.664,38.383,157.241
C02507=1043.814,172.992,404.278,170.666,38.385,157.242
C02508=1043.821,173.277,404.250,170.668,38.386,157.242
C02509=1043.828,173.561,404.225,170.672,38.387,157.243
C02510=1043.834,173.846,404.198,170.674,38.389,157.243
C02511=1043.842,174.131,404.171,170.677,38.391,157.243
C02512=1043.848,174.380,404.148,170.680,38.392,157.244
C02513=1043.854,174.628,404.125,170.682,38.394,157.244
C02514=1043.860,174.878,404.101,170.684,38.395,157.244
C02515=1043.866,175.127,404.078,170.688,38.397,157.245
C02516=1043.872,175.375,404.055,170.690,38.398,157.245
C02517=1043.878,175.625,404.032,170.692,38.400,157.245
C02518=1043.885,175.873,404.008,170.694,38.401,157.246
C02519=1043.891,176.121,403.985,170.697,38.402,157.246
C02520=1043.897,176.371,403.962,170.699,38.404,157.246
C02521=1043.903,176.619,403.939,170.702,38.405,157.247
C02522=1043.909,176.868,403.916,170.704,38.406,157.247
C02523=1043.916,177.117,403.892,170.707,38.408,157.247
C02524=1043.921,177.366,403.869,170.709,38.409,157.248
C02525=1043.928,177.615,403.845,170.711,38.410,157.248
C02526=1043.934,177.864,403.822,170.715,38.412,157.248
C02527=1043.940,178.112,403.798,170.717,38.413,157.249
C02528=1043.947,178.361,403.775,170.719,38.415,157.249
C02529=1043.953,178.610,403.752,170.721,38.416,157.249
C02530=1043.959,178.859,403.728,170.724,38.418,157.250
C02531=1043.965,179.108,403.705,170.727,38.419,157.250
C02532=1043.971,179.356,403.681,170.729,38.421,157.250
C02533=1043.978,179.605,403.658,170.732,38.422,157.251
C02534=1043.984,179.854,403.634,170.734,38.424,157.251
C02535=1043.990,180.103,403.611,170.737,38.425,157.251
C02536=1043.996,180.352,403.587,170.740,38.427,157.252
C02537=1044.003,180.601,403.563,170.742,38.428,157.252
C02538=1044.008,180.850,403.540,170.744,38.429,157.253
C02539=1044.015,181.099,403.516,170.747,38.431,157.253
C02540=1044.022,181.347,403.494,170.750,38.432,157.253
C02541=1044.028,181.596,403.470,170.752,38.433,157.254
C02542=1044.034,181.844,403.446,170.754,38.435,157.254
C02543=1044.041,182.094,403.423,170.758,38.436,157.254
C02544=1044.047,182.342,403.399,170.760,38.438,157.255
C02545=1044.053,182.591,403.375,170.762,38.439,157.255
C02546=1044.059,182.840,403.352,170.764,38.441,157.255
C02547=1044.066,183.089,403.328,170.768,38.442,157.256
C02548=1044.072,183.337,403.304,170.770,38.444,157.256
C02549=1044.078,183.586,403.280,170.772,38.445,157.256
C02550=1044.084,183.835,403.257,170.775,38.447,157.257
C02551=1044.090,184.085,403.233,170.778,38.448,157.257
C02552=1044.096,184.333,403.209,170.780,38.449,157.257
C02553=1044.102,184.581,403.185,170.783,38.451,157.258
C02554=1044.108,184.830,403.161,170.785,38.453,157.258
C02555=1044.114,185.079,403.137,170.787,38.455,157.259
C02556=1044.120,185.328,403.113,170.791,38.456,157.259
C02557=1044.126,185.576,403.089,170.793,38.458,157.259
C02558=1044.132,185.825,403.064,170.795,38.459,157.260
C02559=1044.138,186.074,403.041,170.798,38.461,157.260
C02560=1044.143,186.322,403.016,170.801,38.463,157.260
C02561=1044.150,186.571,402.992,170.803,38.464,157.261
C02562=1044.155,186.820,402.968,170.806,38.466,157.261
C02563=1044.162,187.069,402.944,170.808,38.467,157.262
C02564=1044.167,187.317,402.920,170.811,38.469,157.262
C02565=1044.174,187.566,402.896,170.813,38.471,157.262
C02566=1044.179,187.815,402.871,170.816,38.473,157.263
C02567=1044.186,188.064,402.847,170.818,38.474,157.263
C02568=1044.191,188.313,402.823,170.822,38.476,157.264
C02569=1044.198,188.562,402.799,170.824,38.477,157.264
C02570=1044.203,188.810,402.775,170.826,38.479,157.264
C02571=1044.209,189.059,402.751,170.828,38.481,157.265
C02572=1044.216,189.344,402.723,170.832,38.482,157.265
C02573=1044.223,189.628,402.695,170.835,38.485,157.266
C02574=1044.230,189.913,402.668,170.838,38.486,157.266
C02575=1044.237,190.197,402.640,170.841,38.488,157.266
C02576=1044.242,190.445,402.616,170.843,38.490,157.267
C02577=1044.249,190.694,402.591,170.846,38.492,157.267
C02578=1044.255,190.944,402.567,170.849,38.493,157.268
C02579=1044.261,191.192,402.543,170.851,38.495,157.268
C02580=1044.267,191.441,402.518,170.854,38.497,157.269
C02581=1044.273,191.689,402.494,170.857,38.498,157.269
C02582=1044.279,191.938,402.470,170.859,38.500,157.269
C02583=1044.286,192.187,402.446,170.862,38.501,157.270
C02584=1044.291,192.436,402.421,170.864,38.503,157.270
C02585=1044.298,192.684,402.397,170.867,38.505,157.270
C02586=1044.303,192.933,402.372,170.870,38.506,157.271
C02587=1044.310,193.182,402.348,170.872,38.508,157.271
C02588=1044.316,193.431,402.324,170.875,38.510,157.272
C02589=1044.322,193.679,402.299,170.878,38.512,157.272
C02590=1044.328,193.928,402.275,170.880,38.513,157.272
C02591=1044.334,194.177,402.250,170.883,38.514,157.273
C02592=1044.340,194.425,402.226,170.886,38.516,157.273
C02593=1044.346,194.674,402.201,170.888,38.518,157.274
C02594=1044.353,194.923,402.177,170.891,38.520,157.274
C02595=1044.358,195.171,402.152,170.894,38.521,157.274
C02596=1044.365,195.420,402.128,170.896,38.523,157.275
C02597=1044.371,195.669,402.103,170.900,38.525,157.275
C02598=1044.377,195.917,402.079,170.902,38.527,157.276
C02599=1044.383,196.166,402.054,170.904,38.528,157.276
C02600=1044.389,196.416,402.030,170.908,38.530,157.276
C02601=1044.396,196.664,402.005,170.910,38.532,157.277
C02602=1044.401,196.913,401.981,170.913,38.533,157.277
C02603=1044.408,197.161,401.956,170.916,38.535,157.278
C02604=1044.414,197.410,401.931,170.918,38.536,157.278
C02605=1044.421,197.659,401.907,170.921,38.538,157.278
C02606=1044.426,197.907,401.882,170.924,38.540,157.279
C02607=1044.432,198.157,401.858,170.926,38.541,157.279
C02608=1044.439,198.405,401.833,170.929,38.543,157.280
C02609=1044.445,198.654,401.808,170.932,38.545,157.280
C02610=1044.451,198.902,401.784,170.935,38.547,157.280
C02611=1044.457,199.151,401.759,170.937,38.548,157.281
C02612=1044.463,199.400,401.734,170.940,38.550,157.281
C02613=1044.470,199.649,401.710,170.943,38.552,157.282
C02614=1044.476,199.897,401.685,170.945,38.553,157.282
C02615=1044.483,200.145,401.660,170.949,38.555,157.283
C02616=1044.489,200.394,401.636,170.951,38.557,157.283
C02617=1044.495,200.643,401.610,170.955,38.559,157.283
C02618=1044.501,200.892,401.586,170.957,38.560,157.284
C02619=1044.508,201.141,401.561,170.959,38.562,157.284
C02620=1044.514,201.390,401.537,170.963,38.564,157.285
C02621=1044.520,201.638,401.512,170.965,38.565,157.285
C02622=1044.526,201.886,401.487,170.968,38.568,157.286
C02623=1044.532,202.135,401.461,170.971,38.569,157.286
C02624=1044.538,202.384,401.437,170.973,38.571,157.286
C02625=1044.544,202.633,401.411,170.976,38.573,157.287
C02626=1044.551,202.882,401.386,170.979,38.575,157.287
C02627=1044.556,203.130,401.361,170.982,38.577,157.288
C02628=1044.562,203.379,401.336,170.985,38.579,157.288
C02629=1044.568,203.628,401.311,170.987,38.580,157.289
C02630=1044.575,203.876,401.286,170.990,38.582,157.289
C02631=1044.581,204.125,401.260,170.993,38.584,157.289
C02632=1044.587,204.374,401.236,170.996,38.586,157.290
C02633=1044.593,204.622,401.211,170.999,38.588,157.290
C02634=1044.599,204.870,401.186,171.002,38.589,157.291
C02635=1044.605,205.119,401.161,171.004,38.591,157.291
C02636=1044.631,206.171,401.054,171.266,38.692,157.318
C02637=1044.638,206.453,401.024,171.268,38.695,157.319
C02638=1044.646,206.734,400.994,171.271,38.698,157.320
C02639=1044.654,207.016,400.964,171.273,38.701,157.320
C02640=1044.661,207.298,400.935,171.275,38.704,157.321
C02641=1044.668,207.546,400.909,171.277,38.707,157.322
C02642=1044.675,207.795,400.883,171.279,38.710,157.322
C02643=1044.680,208.043,400.856,171.282,38.712,157.323
C02644=1044.688,208.292,400.830,171.284,38.715,157.323
C02645=1044.694,208.540,400.804,171.286,38.717,157.324
C02646=1044.700,208.789,400.777,171.288,38.720,157.325
C02647=1044.707,209.037,400.751,171.290,38.723,157.325
C02648=1044.714,209.286,400.724,171.292,38.725,157.326
C02649=1044.720,209.534,400.698,171.294,38.728,157.326
C02650=1044.727,209.783,400.671,171.296,38.730,157.327
C02651=1044.733,210.031,400.645,171.299,38.733,157.328
C02652=1044.740,210.280,400.618,171.300,38.735,157.328
C02653=1044.747,210.529,400.592,171.303,38.738,157.329
C02654=1044.753,210.777,400.566,171.304,38.741,157.329
C02655=1044.760,211.026,400.538,171.307,38.743,157.330
C02656=1044.767,211.274,400.512,171.310,38.746,157.331
C02657=1044.773,211.523,400.485,171.311,38.748,157.331
C02658=1044.780,211.771,400.459,171.314,38.751,157.332
C02659=1044.786,212.020,400.432,171.315,38.754,157.332
C02660=1044.792,212.268,400.406,171.318,38.757,157.333
C02661=1044.799,212.517,400.379,171.320,38.759,157.334
C02662=1044.805,212.765,400.353,171.322,38.762,157.334
C02663=1044.812,213.013,400.325,171.324,38.764,157.335
C02664=1044.819,213.262,400.298,171.326,38.767,157.335
C02665=1044.825,213.510,400.272,171.328,38.770,157.336
C02666=1044.832,213.759,400.245,171.331,38.772,157.336
C02667=1044.838,214.008,400.219,171.332,38.775,157.337
C02668=1044.844,214.256,400.191,171.335,38.777,157.338
C02669=1044.851,214.504,400.165,171.337,38.780,157.338
C02670=1044.857,214.753,400.138,171.339,38.783,157.339
C02671=1044.864,215.002,400.112,171.342,38.785,157.340
C02672=1044.871,215.250,400.084,171.343,38.788,157.340
C02673=1044.878,215.498,400.058,171.346,38.790,157.341
C02674=1044.883,215.747,400.031,171.348,38.793,157.341
C02675=1044.891,215.995,400.005,171.350,38.795,157.342
C02676=1044.897,216.244,399.977,171.352,38.798,157.343
C02677=1044.903,216.492,399.950,171.355,38.801,157.343
C02678=1044.910,216.741,399.924,171.356,38.803,157.344
C02679=1044.917,216.989,399.896,171.359,38.806,157.344
C02680=1044.923,217.238,399.870,171.361,38.808,157.345
C02681=1044.930,217.487,399.843,171.363,38.811,157.346
C02682=1044.936,217.735,399.815,171.366,38.814,157.346
C02683=1044.943,217.983,399.789,171.368,38.816,157.347
C02684=1044.950,218.232,399.762,171.370,38.819,157.347
C02685=1044.957,218.480,399.735,171.372,38.821,157.348
C02686=1044.962,218.729,399.709,171.375,38.824,157.349
C02687=1044.969,218.977,399.681,171.376,38.827,157.349
C02688=1044.976,219.226,399.654,171.379,38.829,157.350
C02689=1044.982,219.474,399.627,171.381,38.832,157.350
C02690=1044.989,219.722,399.601,171.384,38.834,157.351
C02691=1044.996,219.971,399.574,171.385,38.836,157.351
C02692=1045.002,220.220,399.546,171.388,38.839,157.352
C02693=1045.010,220.507,399.515,171.391,38.842,157.353
C02694=1045.017,220.794,399.484,171.393,38.845,157.353
C02695=1045.025,221.081,399.452,171.396,38.848,157.354
C02696=1045.032,221.368,399.421,171.398,38.851,157.355
C02697=1045.039,221.617,399.393,171.401,38.854,157.355
C02698=1045.045,221.866,399.366,171.403,38.856,157.356
C02699=1045.052,222.113,399.339,171.405,38.859,157.357
C02700=1045.059,222.362,399.312,171.408,38.862,157.357
C02701=1045.065,222.611,399.285,171.409,38.864,157.358
C02702=1045.071,222.858,399.257,171.412,38.867,157.358
C02703=1045.078,223.107,399.230,171.414,38.869,157.359
C02704=1045.084,223.356,399.202,171.417,38.872,157.360
C02705=1045.091,223.604,399.175,171.418,38.874,157.360
C02706=1045.097,223.852,399.149,171.421,38.877,157.361
C02707=1045.104,224.101,399.121,171.424,38.880,157.361
C02708=1045.111,224.349,399.093,171.426,38.882,157.362
C02709=1045.117,224.598,399.066,171.428,38.885,157.363
C02710=1045.123,224.846,399.039,171.430,38.887,157.363
C02711=1045.130,225.094,399.011,171.433,38.890,157.364
C02712=1045.137,225.343,398.983,171.435,38.893,157.364
C02713=1045.143,225.592,398.956,171.437,38.895,157.365
C02714=1045.150,225.840,398.929,171.439,38.898,157.366
C02715=1045.156,226.088,398.902,171.442,38.900,157.366
C02716=1045.163,226.336,398.874,171.444,38.902,157.367
C02717=1045.170,226.585,398.847,171.446,38.905,157.367
C02718=1045.176,226.834,398.819,171.449,38.908,157.368
C02719=1045.183,227.082,398.792,171.451,38.911,157.369
C02720=1045.190,227.331,398.764,171.454,38.913,157.369
C02721=1045.196,227.578,398.737,171.456,38.915,157.370
C02722=1045.202,227.827,398.710,171.458,38.918,157.370
C02723=1045.209,228.076,398.682,171.460,38.920,157.371
C02724=1045.216,228.324,398.655,171.463,38.923,157.372
C02725=1045.223,228.573,398.627,171.465,38.926,157.372
C02726=1045.230,228.821,398.599,171.468,38.928,157.373
C02727=1045.236,229.069,398.571,171.469,38.930,157.373
C02728=1045.242,229.317,398.544,171.472,38.933,157.374
C02729=1045.248,229.566,398.516,171.475,38.936,157.375
C02730=1045.255,229.815,398.489,171.477,38.938,157.375
C02731=1045.261,230.063,398.461,171.480,38.941,157.376
C02732=1045.268,230.312,398.433,171.482,38.944,157.377
C02733=1045.275,230.560,398.406,171.484,38.946,157.377
C02734=1045.281,230.809,398.378,171.486,38.948,157.378
C02735=1045.287,231.056,398.351,171.489,38.951,157.378
C02736=1045.294,231.305,398.323,171.492,38.954,157.379
C02737=1045.301,231.553,398.295,171.494,38.956,157.380
C02738=1045.307,231.802,398.267,171.496,38.959,157.380
C02739=1045.313,232.051,398.239,171.498,38.962,157.381
C02740=1045.320,232.298,398.211,171.501,38.964,157.381
C02741=1045.327,232.547,398.183,171.503,38.966,157.382
C02742=1045.334,232.795,398.155,171.506,38.969,157.383
C02743=1045.340,233.044,398.127,171.508,38.972,157.383
C02744=1045.346,233.292,398.099,171.511,38.974,157.384
C02745=1045.352,233.540,398.072,171.513,38.977,157.384
C02746=1045.359,233.789,398.044,171.515,38.980,157.385
C02747=1045.365,234.037,398.016,171.518,38.982,157.386
C02748=1045.372,234.285,397.987,171.520,38.985,157.386
C02749=1045.379,234.565,397.956,171.523,38.988,157.387
C02750=1045.387,234.845,397.925,171.526,38.991,157.388
C02751=1045.394,235.124,397.893,171.528,38.994,157.388
C02752=1045.401,235.404,397.861,171.531,38.996,157.389
C02753=1045.408,235.653,397.833,171.533,38.999,157.390
C02754=1045.414,235.901,397.806,171.536,39.001,157.390
C02755=1045.421,236.149,397.777,171.539,39.004,157.391
C02756=1045.427,236.398,397.749,171.541,39.006,157.391
C02757=1045.434,236.646,397.721,171.544,39.009,157.392
C02758=1045.441,236.894,397.693,171.546,39.011,157.393
C02759=1045.447,237.143,397.664,171.549,39.014,157.393
C02760=1045.454,237.391,397.637,171.551,39.017,157.394
C02761=1045.460,237.640,397.609,171.553,39.019,157.394
C02762=1045.467,237.887,397.580,171.556,39.022,157.395
C02763=1045.473,238.136,397.552,171.558,39.024,157.396
C02764=1045.480,238.385,397.524,171.561,39.026,157.396
C02765=1045.487,238.632,397.496,171.563,39.029,157.397
C02766=1045.493,238.881,397.468,171.566,39.032,157.397
C02767=1045.499,239.130,397.440,171.568,39.035,157.398
C02768=1045.506,239.377,397.411,171.571,39.037,157.399
C02769=1045.512,239.626,397.383,171.574,39.040,157.399
C02770=1045.519,239.874,397.355,171.576,39.042,157.400
C02771=1045.525,240.123,397.326,171.579,39.044,157.401
C02772=1045.532,240.370,397.298,171.581,39.047,157.401
C02773=1045.540,240.620,397.270,171.584,39.049,157.402
C02774=1045.546,240.868,397.241,171.586,39.052,157.402
C02775=1045.552,241.116,397.213,171.589,39.055,157.403
C02776=1045.559,241.365,397.185,171.590,39.057,157.404
C02777=1045.565,241.613,397.156,171.593,39.060,157.404
C02778=1045.572,241.861,397.127,171.596,39.062,157.405
C02779=1045.578,242.109,397.099,171.598,39.065,157.405
C02780=1045.585,242.357,397.070,171.601,39.067,157.406
C02781=1045.591,242.606,397.043,171.603,39.070,157.407
C02782=1045.598,242.854,397.014,171.606,39.073,157.407
C02783=1045.604,243.102,396.985,171.609,39.075,157.408
C02784=1045.610,243.351,396.957,171.611,39.078,157.409
C02785=1045.617,243.599,396.928,171.614,39.081,157.409
C02786=1045.624,243.848,396.900,171.616,39.083,157.410
C02787=1045.630,244.096,396.871,171.619,39.086,157.410
C02788=1045.636,244.344,396.842,171.621,39.088,157.411
C02789=1045.643,244.593,396.814,171.624,39.091,157.412
C02790=1045.649,244.841,396.785,171.627,39.093,157.412
C02791=1045.656,245.089,396.756,171.629,39.096,157.413
C02792=1045.663,245.337,396.727,171.632,39.098,157.414
C02793=1045.669,245.585,396.699,171.634,39.101,157.414
C02794=1045.675,245.834,396.670,171.637,39.104,157.415
C02795=1045.682,246.082,396.641,171.640,39.106,157.415
C02796=1045.689,246.330,396.612,171.642,39.109,157.416
C02797=1045.695,246.578,396.583,171.645,39.112,157.417
C02798=1045.701,246.827,396.555,171.647,39.114,157.417
C02799=1045.707,247.075,396.526,171.650,39.117,157.418
C02800=1045.713,247.323,396.497,171.653,39.120,157.419
C02801=1045.720,247.572,396.468,171.655,39.122,157.419
C02802=1045.727,247.819,396.439,171.658,39.125,157.420
C02803=1045.733,248.067,396.410,171.660,39.127,157.421
C02804=1045.740,248.316,396.381,171.663,39.130,157.421
C02805=1045.747,248.590,396.349,171.666,39.133,157.422
C02806=1045.753,248.864,396.317,171.668,39.136,157.423
C02807=1045.760,249.138,396.285,171.672,39.139,157.423
C02808=1045.768,249.411,396.253,171.675,39.141,157.424
C02809=1045.774,249.660,396.225,171.677,39.144,157.425
C02810=1045.781,249.909,396.195,171.680,39.147,157.425
C02811=1045.787,250.157,396.166,171.682,39.149,157.426
C02812=1045.793,250.405,396.137,171.685,39.152,157.426
C02813=1045.799,250.653,396.108,171.688,39.155,157.427
C02814=1045.806,250.901,396.078,171.690,39.157,157.428
C02815=1045.813,251.149,396.050,171.693,39.160,157.428
C02816=1045.820,251.397,396.021,171.695,39.162,157.429
C02817=1045.826,251.646,395.991,171.698,39.165,157.430
C02818=1045.832,251.894,395.962,171.701,39.168,157.430
C02819=1045.839,252.142,395.933,171.703,39.170,157.431
C02820=1045.845,252.391,395.904,171.707,39.173,157.432
C02821=1045.852,252.639,395.875,171.709,39.175,157.432
C02822=1045.858,252.887,395.846,171.712,39.178,157.433
C02823=1045.865,253.136,395.816,171.714,39.180,157.433
C02824=1045.871,253.384,395.787,171.717,39.183,157.434
C02825=1045.878,253.631,395.758,171.720,39.185,157.435
C02826=1045.885,253.880,395.729,171.722,39.188,157.435
C02827=1045.891,254.128,395.700,171.725,39.191,157.436
C02828=1045.898,254.376,395.671,171.728,39.193,157.437
C02829=1045.904,254.625,395.641,171.730,39.196,157.437
C02830=1045.911,254.872,395.612,171.734,39.199,157.438
C02831=1045.917,255.121,395.583,171.736,39.201,157.439
C02832=1045.924,255.369,395.553,171.739,39.204,157.439
C02833=1045.930,255.618,395.524,171.742,39.207,157.440
C02834=1045.937,255.866,395.495,171.744,39.209,157.441
C02835=1045.944,256.114,395.465,171.747,39.212,157.441
C02836=1045.950,256.362,395.436,171.749,39.214,157.442
C02837=1045.957,256.610,395.408,171.753,39.217,157.442
C02838=1045.964,256.858,395.377,171.756,39.219,157.443
C02839=1045.970,257.106,395.348,171.758,39.222,157.444
C02840=1045.977,257.355,395.319,171.761,39.224,157.444
C02841=1045.984,257.603,395.289,171.763,39.227,157.445
C02842=1045.990,257.851,395.260,171.766,39.229,157.446
C02843=1045.997,258.100,395.231,171.770,39.232,157.446
C02844=1046.003,258.347,395.201,171.772,39.234,157.447
C02845=1046.010,258.596,395.172,171.775,39.237,157.448
C02846=1046.017,258.844,395.143,171.777,39.239,157.448
C02847=1046.024,259.092,395.112,171.780,39.242,157.449
C02848=1046.030,259.340,395.083,171.783,39.245,157.449
C02849=1046.036,259.588,395.054,171.786,39.247,157.450
C02850=1046.043,259.837,395.024,171.789,39.250,157.451
C02851=1046.050,260.084,394.994,171.791,39.252,157.451
C02852=1046.057,260.333,394.965,171.794,39.255,157.452
C02853=1046.063,260.581,394.935,171.798,39.258,157.453
C02854=1046.070,260.829,394.906,171.800,39.260,157.453
C02855=1046.077,261.077,394.876,171.803,39.263,157.454
C02856=1046.084,261.326,394.847,171.805,39.265,157.454
C02857=1046.090,261.573,394.817,171.808,39.268,157.455
C02858=1046.097,261.822,394.788,171.812,39.270,157.456
C02859=1046.104,262.070,394.758,171.814,39.273,157.456
C02860=1046.110,262.318,394.728,171.817,39.275,157.457
C02861=1046.118,262.590,394.696,171.820,39.278,157.458
C02862=1046.125,262.862,394.663,171.823,39.281,157.458
C02863=1046.132,263.135,394.630,171.826,39.284,157.459
C02864=1046.140,263.408,394.598,171.830,39.287,157.460
C02865=1046.146,263.656,394.567,171.832,39.289,157.461
C02866=1046.153,263.904,394.537,171.835,39.292,157.461
C02867=1046.159,264.152,394.508,171.838,39.295,157.462
C02868=1046.165,264.401,394.477,171.841,39.297,157.463
C02869=1046.172,264.648,394.448,171.844,39.300,157.463
C02870=1046.179,264.896,394.418,171.846,39.303,157.464
C02871=1046.185,265.144,394.387,171.849,39.305,157.465
C02872=1046.192,265.393,394.358,171.853,39.308,157.465
C02873=1046.198,265.640,394.328,171.855,39.311,157.466
C02874=1046.205,265.889,394.297,171.858,39.313,157.466
C02875=1046.211,266.136,394.268,171.861,39.316,157.467
C02876=1046.219,266.385,394.237,171.864,39.319,157.468
C02877=1046.224,266.633,394.207,171.867,39.321,157.468
C02878=1046.231,266.881,394.178,171.869,39.324,157.469
C02879=1046.238,267.130,394.147,171.873,39.326,157.470
C02880=1046.244,267.377,394.117,171.876,39.329,157.470
C02881=1046.251,267.626,394.087,171.878,39.332,157.471
C02882=1046.257,267.873,394.057,171.881,39.334,157.472
C02883=1046.264,268.122,394.027,171.885,39.337,157.473
C02884=1046.270,268.369,393.996,171.887,39.339,157.473
C02885=1046.277,268.618,393.966,171.890,39.342,157.474
C02886=1046.284,268.866,393.935,171.894,39.345,157.475
C02887=1046.290,269.114,393.906,171.896,39.347,157.475
C02888=1046.297,269.362,393.875,171.899,39.350,157.476
C02889=1046.303,269.610,393.845,171.902,39.353,157.477
C02890=1046.310,269.858,393.814,171.905,39.356,157.477
C02891=1046.317,270.106,393.784,171.908,39.358,157.478
C02892=1046.323,270.354,393.754,171.910,39.361,157.479
C02893=1046.330,270.603,393.724,171.914,39.364,157.479
C02894=1046.336,270.850,393.692,171.917,39.367,157.480
C02895=1046.343,271.098,393.663,171.919,39.369,157.481
C02896=1046.349,271.346,393.632,171.923,39.372,157.481
C02897=1046.357,271.595,393.602,171.926,39.374,157.482
C02898=1046.362,271.842,393.571,171.928,39.377,157.483
C02899=1046.370,272.091,393.541,171.932,39.379,157.483
C02900=1046.376,272.339,393.510,171.935,39.382,157.484
C02901=1046.382,272.586,393.480,171.937,39.385,157.485
C02902=1046.389,272.835,393.449,171.941,39.388,157.485
C02903=1046.396,273.083,393.419,171.944,39.391,157.486
C02904=1046.402,273.330,393.388,171.946,39.393,157.487
C02905=1046.409,273.579,393.358,171.950,39.396,157.487
C02906=1046.415,273.827,393.327,171.953,39.399,157.488
C02907=1046.422,274.074,393.296,171.956,39.401,157.489
C02908=1046.429,274.323,393.266,171.959,39.404,157.490
C02909=1046.435,274.571,393.235,171.961,39.406,157.490
C02910=1046.441,274.818,393.204,171.965,39.409,157.491
C02911=1046.448,275.066,393.174,171.968,39.412,157.492
C02912=1046.455,275.315,393.143,171.971,39.415,157.492
C02913=1046.462,275.563,393.112,171.974,39.418,157.493
C02914=1046.467,275.811,393.081,171.977,39.420,157.494
C02915=1046.474,276.059,393.050,171.981,39.423,157.494
C02916=1046.481,276.307,393.020,171.983,39.425,157.495
C02917=1046.488,276.584,392.985,171.987,39.429,157.496
C02918=1046.496,276.861,392.951,171.990,39.432,157.497
C02919=1046.503,277.137,392.916,171.994,39.435,157.497
C02920=1046.510,277.414,392.882,171.997,39.438,157.498
C02921=1046.517,277.662,392.851,172.000,39.441,157.499
C02922=1046.524,277.910,392.820,172.003,39.443,157.500
C02923=1046.530,278.158,392.790,172.006,39.446,157.500
C02924=1046.537,278.406,392.758,172.009,39.449,157.501
C02925=1046.544,278.654,392.727,172.013,39.451,157.502
C02926=1046.550,278.902,392.696,172.015,39.454,157.502
C02927=1046.557,279.150,392.665,172.019,39.457,157.503
C02928=1046.564,279.398,392.635,172.022,39.460,157.504
C02929=1046.570,279.645,392.604,172.024,39.462,157.504
C02930=1046.577,279.893,392.572,172.028,39.465,157.505
C02931=1046.583,280.142,392.541,172.031,39.468,157.506
C02932=1046.590,280.390,392.510,172.034,39.471,157.507
C02933=1046.597,280.638,392.479,172.037,39.474,157.507
C02934=1046.603,280.885,392.448,172.041,39.476,157.508
C02935=1046.609,281.133,392.417,172.044,39.479,157.509
C02936=1046.616,281.381,392.385,172.047,39.482,157.509
C02937=1046.623,281.629,392.354,172.050,39.485,157.510
C02938=1046.629,281.877,392.323,172.053,39.488,157.511
C02939=1046.635,282.125,392.291,172.056,39.490,157.512
C02940=1046.642,282.374,392.260,172.059,39.493,157.512
C02941=1046.648,282.621,392.229,172.063,39.496,157.513
C02942=1046.655,282.869,392.197,172.065,39.499,157.514
C02943=1046.661,283.117,392.166,172.069,39.501,157.514
C02944=1046.668,283.365,392.134,172.072,39.504,157.515
C02945=1046.675,283.613,392.103,172.076,39.507,157.516
C02946=1046.681,283.861,392.072,172.078,39.510,157.517
C02947=1046.688,284.109,392.041,172.082,39.513,157.517
C02948=1046.695,284.357,392.009,172.085,39.515,157.518
C02949=1046.701,284.605,391.978,172.088,39.518,157.519
C02950=1046.708,284.853,391.947,172.091,39.521,157.520
C02951=1046.715,285.101,391.915,172.095,39.524,157.520
C02952=1046.721,285.349,391.884,172.097,39.527,157.521
C02953=1046.728,285.596,391.852,172.101,39.529,157.522
C02954=1046.735,285.844,391.821,172.104,39.532,157.522
C02955=1046.742,286.092,391.789,172.108,39.535,157.523
C02956=1046.748,286.340,391.758,172.111,39.538,157.524
C02957=1046.755,286.588,391.727,172.114,39.540,157.525
C02958=1046.762,286.836,391.695,172.118,39.543,157.525
C02959=1046.769,287.083,391.663,172.120,39.546,157.526
C02960=1046.776,287.331,391.632,172.124,39.549,157.527
C02961=1046.782,287.579,391.599,172.127,39.552,157.527
C02962=1046.788,287.827,391.568,172.130,39.554,157.528
C02963=1046.795,288.075,391.537,172.133,39.558,157.529
C02964=1046.802,288.323,391.505,172.137,39.560,157.530
C02965=1046.808,288.571,391.473,172.141,39.563,157.530
C02966=1046.815,288.819,391.441,172.143,39.566,157.531
C02967=1046.822,289.067,391.410,172.147,39.569,157.532
C02968=1046.828,289.314,391.378,172.150,39.571,157.533
C02969=1046.834,289.563,391.346,172.154,39.574,157.533
C02970=1046.841,289.810,391.314,172.156,39.578,157.534
C02971=1046.848,290.058,391.283,172.160,39.580,157.535
C02972=1046.855,290.306,391.251,172.164,39.583,157.536
C02973=1046.862,290.595,391.213,172.168,39.586,157.537
C02974=1046.870,290.882,391.177,172.172,39.590,157.537
C02975=1046.878,291.171,391.139,172.175,39.593,157.538
C02976=1046.885,291.459,391.102,172.179,39.596,157.539
C02977=1046.892,291.707,391.070,172.182,39.599,157.540
C02978=1046.898,291.955,391.038,172.186,39.602,157.541
C02979=1046.905,292.202,391.006,172.189,39.605,157.541
C02980=1046.912,292.451,390.974,172.192,39.608,157.542
C02981=1046.919,292.699,390.942,172.196,39.611,157.543
C02982=1046.926,292.946,390.910,172.199,39.614,157.544
C02983=1046.932,293.194,390.878,172.203,39.617,157.545
C02984=1046.939,293.442,390.846,172.206,39.620,157.545
C02985=1046.946,293.690,390.814,172.209,39.622,157.546
C02986=1046.952,293.937,390.782,172.213,39.625,157.547
C02987=1046.959,294.185,390.749,172.217,39.628,157.548
C02988=1046.965,294.433,390.717,172.219,39.631,157.548
C02989=1046.972,294.681,390.685,172.223,39.634,157.549
C02990=1046.978,294.929,390.653,172.226,39.637,157.550
C02991=1046.986,295.176,390.621,172.230,39.640,157.551
C02992=1046.992,295.424,390.588,172.233,39.643,157.551
C02993=1046.999,295.672,390.556,172.236,39.646,157.552
C02994=1047.005,295.920,390.524,172.240,39.649,157.553
C02995=1047.012,296.167,390.491,172.244,39.652,157.554
C02996=1047.018,296.415,390.459,172.246,39.655,157.555
C02997=1047.025,296.663,390.427,172.250,39.658,157.555
C02998=1047.031,296.911,390.394,172.254,39.661,157.556
C02999=1047.039,297.159,390.361,172.257,39.664,157.557
C03000=1047.045,297.406,390.329,172.260,39.667,157.558
C03001=1047.051,297.654,390.296,172.264,39.670,157.558
C03002=1047.057,297.902,390.264,172.267,39.673,157.559
C03003=1047.064,298.150,390.231,172.271,39.676,157.560
C03004=1047.071,298.398,390.199,172.275,39.679,157.561
C03005=1047.077,298.645,390.166,172.278,39.682,157.562
C03006=1047.084,298.893,390.133,172.281,39.685,157.562
C03007=1047.090,299.140,390.100,172.285,39.688,157.563
C03008=1047.097,299.389,390.067,172.288,39.691,157.564
C03009=1047.104,299.636,390.035,172.292,39.694,157.565
C03010=1047.110,299.884,390.002,172.295,39.697,157.566
C03011=1047.117,300.131,389.970,172.299,39.700,157.566
C03012=1047.123,300.379,389.937,172.302,39.703,157.567
C03013=1047.130,300.627,389.904,172.306,39.706,157.568
C03014=1047.137,300.874,389.872,172.310,39.709,157.569
C03015=1047.143,301.122,389.839,172.312,39.713,157.570
C03016=1047.150,301.370,389.806,172.316,39.716,157.571
C03017=1047.156,301.618,389.773,172.320,39.719,157.571
C03018=1047.163,301.865,389.740,172.324,39.722,157.572
C03019=1047.169,302.114,389.707,172.327,39.725,157.573
C03020=1047.177,302.360,389.674,172.331,39.728,157.574
C03021=1047.183,302.608,389.642,172.334,39.731,157.575
C03022=1047.190,302.856,389.609,172.338,39.734,157.575
C03023=1047.196,303.104,389.576,172.342,39.737,157.576
C03024=1047.203,303.352,389.543,172.345,39.740,157.577
C03025=1047.210,303.599,389.509,172.349,39.743,157.578
C03026=1047.217,303.846,389.477,172.352,39.746,157.579
C03027=1047.224,304.095,389.444,172.356,39.749,157.579
C03028=1047.230,304.342,389.411,172.359,39.752,157.580
C03029=1047.239,304.647,389.370,172.364,39.756,157.581
C03030=1047.247,304.951,389.330,172.368,39.760,157.582
C03031=1047.255,305.256,389.289,172.373,39.764,157.583
C03032=1047.263,305.561,389.248,172.377,39.767,157.584
C03033=1047.270,305.808,389.216,172.381,39.771,157.585
C03034=1047.277,306.056,389.182,172.385,39.773,157.586
C03035=1047.284,306.303,389.150,172.389,39.777,157.587
C03036=1047.291,306.551,389.116,172.392,39.780,157.588
C03037=1047.297,306.799,389.083,172.395,39.783,157.588
C03038=1047.304,307.047,389.050,172.399,39.786,157.589
C03039=1047.311,307.294,389.017,172.403,39.789,157.590
C03040=1047.318,307.542,388.983,172.407,39.792,157.591
C03041=1047.324,307.789,388.950,172.411,39.795,157.592
C03042=1047.331,308.037,388.917,172.414,39.798,157.593
C03043=1047.338,308.284,388.883,172.418,39.801,157.593
C03044=1047.345,308.532,388.851,172.421,39.805,157.594
C03045=1047.353,308.780,388.817,172.425,39.808,157.595
C03046=1047.359,309.028,388.784,172.429,39.811,157.596
C03047=1047.366,309.275,388.751,172.433,39.814,157.597
C03048=1047.372,309.523,388.718,172.436,39.817,157.598
C03049=1047.380,309.771,388.684,172.440,39.820,157.598
C03050=1047.387,310.018,388.650,172.444,39.823,157.599
C03051=1047.393,310.266,388.617,172.448,39.826,157.600
C03052=1047.400,310.514,388.584,172.452,39.830,157.601
C03053=1047.407,310.761,388.550,172.456,39.832,157.602
C03054=1047.414,311.009,388.518,172.458,39.836,157.603
C03055=1047.422,311.256,388.484,172.462,39.839,157.604
C03056=1047.429,311.504,388.450,172.466,39.842,157.604
C03057=1047.435,311.751,388.417,172.470,39.845,157.605
C03058=1047.442,311.999,388.383,172.474,39.848,157.606
C03059=1047.450,312.247,388.350,172.478,39.852,157.607
C03060=1047.456,312.494,388.317,172.482,39.855,157.608
C03061=1047.463,312.742,388.283,172.485,39.857,157.609
C03062=1047.470,312.990,388.249,172.489,39.861,157.610
C03063=1047.476,313.237,388.215,172.493,39.864,157.610
C03064=1047.483,313.485,388.181,172.497,39.867,157.611
C03065=1047.490,313.733,388.147,172.501,39.871,157.612
C03066=1047.496,313.980,388.113,172.505,39.874,157.613
C03067=1047.503,314.228,388.079,172.508,39.878,157.614
C03068=1047.510,314.475,388.045,172.512,39.881,157.615
C03069=1047.516,314.723,388.011,172.516,39.884,157.616
C03070=1047.523,314.970,387.977,172.520,39.888,157.617
C03071=1047.530,315.218,387.943,172.524,39.891,157.618
C03072=1047.536,315.465,387.909,172.527,39.894,157.618
C03073=1047.543,315.713,387.875,172.531,39.897,157.619
C03074=1047.550,315.961,387.841,172.535,39.901,157.620
C03075=1047.556,316.208,387.806,172.539,39.904,157.621
C03076=1047.563,316.455,387.773,172.543,39.908,157.622
C03077=1047.570,316.703,387.738,172.547,39.911,157.623
C03078=1047.577,316.951,387.704,172.551,39.914,157.624
C03079=1047.583,317.198,387.670,172.555,39.918,157.625
C03080=1047.590,317.446,387.636,172.559,39.921,157.626
C03081=1047.597,317.693,387.601,172.563,39.924,157.627
C03082=1047.604,317.941,387.568,172.567,39.928,157.628
C03083=1047.610,318.189,387.533,172.571,39.931,157.629
C03084=1047.617,318.436,387.500,172.575,39.934,157.629
C03085=1047.626,318.745,387.456,172.580,39.939,157.631
C03086=1047.634,319.054,387.413,172.584,39.943,157.632
C03087=1047.642,319.364,387.370,172.589,39.947,157.633
C03088=1047.652,319.672,387.328,172.594,39.951,157.634
C03089=1047.658,319.920,387.293,172.598,39.955,157.635
C03090=1047.664,320.168,387.259,172.602,39.958,157.636
C03091=1047.672,320.415,387.225,172.606,39.962,157.637
C03092=1047.678,320.663,387.190,172.610,39.965,157.638
C03093=1047.686,320.910,387.156,172.614,39.968,157.639
C03094=1047.692,321.158,387.121,172.618,39.971,157.640
C03095=1047.699,321.405,387.087,172.622,39.975,157.641
C03096=1047.706,321.653,387.052,172.626,39.978,157.641
C03097=1047.713,321.900,387.018,172.630,39.982,157.642
C03098=1047.720,322.148,386.983,172.634,39.986,157.643
C03099=1047.726,322.396,386.949,172.638,39.989,157.644
C03100=1047.734,322.643,386.914,172.643,39.992,157.645
C03101=1047.741,322.890,386.879,172.647,39.996,157.646
C03102=1047.748,323.138,386.845,172.651,39.999,157.647
C03103=1047.755,323.385,386.810,172.654,40.002,157.648
C03104=1047.762,323.633,386.776,172.658,40.006,157.649
C03105=1047.769,323.880,386.741,172.662,40.009,157.650
C03106=1047.775,324.128,386.706,172.666,40.013,157.651
C03107=1047.783,324.375,386.672,172.670,40.016,157.652
C03108=1047.789,324.623,386.637,172.674,40.020,157.653
C03109=1047.797,324.870,386.603,172.679,40.023,157.654
C03110=1047.803,325.118,386.568,172.683,40.027,157.655
C03111=1047.810,325.365,386.533,172.687,40.030,157.656
C03112=1047.818,325.612,386.498,172.691,40.034,157.657
C03113=1047.825,325.860,386.463,172.695,40.037,157.658
C03114=1047.832,326.108,386.429,172.699,40.041,157.659
C03115=1047.839,326.355,386.394,172.703,40.044,157.659
C03116=1047.846,326.603,386.359,172.708,40.048,157.661
C03117=1047.853,326.850,386.324,172.712,40.051,157.661
C03118=1047.860,327.097,386.289,172.716,40.054,157.662
C03119=1047.867,327.345,386.255,172.720,40.058,157.663
C03120=1047.875,327.593,386.220,172.724,40.061,157.664
C03121=1047.881,327.840,386.185,172.729,40.065,157.665
C03122=1047.888,328.087,386.150,172.733,40.068,157.666
C03123=1047.896,328.334,386.115,172.737,40.072,157.667
C03124=1047.903,328.583,386.080,172.741,40.076,157.668
C03125=1047.911,328.830,386.045,172.745,40.079,157.669
C03126=1047.917,329.077,386.010,172.750,40.083,157.670
C03127=1047.924,329.324,385.975,172.754,40.086,157.671
C03128=1047.932,329.572,385.940,172.758,40.090,157.672
C03129=1047.939,329.819,385.905,172.762,40.094,157.673
C03130=1047.946,330.067,385.870,172.766,40.097,157.674
C03131=1047.952,330.314,385.834,172.771,40.100,157.675
C03132=1047.959,330.561,385.798,172.775,40.104,157.676
C03133=1047.966,330.809,385.763,172.779,40.108,157.677
C03134=1047.973,331.057,385.727,172.783,40.111,157.678
C03135=1047.980,331.304,385.692,172.789,40.115,157.679
C03136=1047.987,331.551,385.656,172.793,40.119,157.680
C03137=1047.994,331.799,385.621,172.797,40.123,157.681
C03138=1048.001,332.046,385.586,172.801,40.126,157.682
C03139=1048.008,332.294,385.551,172.805,40.130,157.683
C03140=1048.015,332.541,385.514,172.810,40.133,157.684
C03141=1048.022,332.763,385.483,172.814,40.137,157.685
C03142=1048.028,332.986,385.451,172.818,40.140,157.686
C03143=1048.034,333.208,385.420,172.822,40.144,157.687
C03144=1048.041,333.430,385.387,172.825,40.147,157.688
C03145=1048.047,333.653,385.355,172.829,40.150,157.689
C03146=1048.053,333.875,385.324,172.833,40.154,157.690
C03147=1048.059,334.097,385.291,172.837,40.157,157.691
C03148=1048.066,334.320,385.259,172.841,40.160,157.692
C03149=1048.073,334.567,385.223,172.846,40.164,157.693
C03150=1048.080,334.815,385.188,172.850,40.168,157.694
C03151=1048.088,335.061,385.152,172.854,40.172,157.695
C03152=1048.094,335.310,385.116,172.859,40.175,157.696
C03153=1048.101,335.556,385.080,172.863,40.179,157.697
C03154=1048.109,335.805,385.045,172.867,40.183,157.698
C03155=1048.116,336.051,385.009,172.872,40.187,157.699
C03156=1048.122,336.299,384.974,172.876,40.190,157.700
C03157=1048.130,336.546,384.937,172.880,40.194,157.701
C03158=1048.136,336.793,384.901,172.884,40.198,157.702
C03159=1048.144,337.041,384.865,172.890,40.202,157.703
C03160=1048.151,337.288,384.830,172.894,40.206,157.705
C03161=1048.158,337.536,384.793,172.898,40.210,157.706
C03162=1048.165,337.782,384.757,172.903,40.213,157.707
C03163=1048.172,338.029,384.721,172.907,40.217,157.708
C03164=1048.179,338.278,384.685,172.912,40.221,157.709
C03165=1048.186,338.524,384.649,172.917,40.225,157.710
C03166=1048.193,338.772,384.613,172.921,40.229,157.711
C03167=1048.200,339.019,384.576,172.926,40.233,157.712
C03168=1048.207,339.266,384.540,172.930,40.237,157.713
C03169=1048.215,339.514,384.504,172.934,40.241,157.714
C03170=1048.221,339.761,384.468,172.939,40.245,157.715
C03171=1048.229,340.008,384.431,172.943,40.248,157.716
C03172=1048.236,340.255,384.395,172.948,40.252,157.718
C03173=1048.243,340.503,384.359,172.953,40.256,157.719
C03174=1048.250,340.750,384.324,172.957,40.260,157.720
C03175=1048.258,340.998,384.287,172.962,40.264,157.721
C03176=1048.265,341.245,384.250,172.966,40.268,157.722
C03177=1048.275,341.599,384.198,172.973,40.274,157.724
C03178=1048.285,341.953,384.146,172.979,40.279,157.725
C03179=1048.296,342.306,384.094,172.986,40.285,157.727
C03180=1048.306,342.660,384.042,172.993,40.291,157.728
C03181=1048.313,342.908,384.005,172.997,40.295,157.730
C03182=1048.320,343.155,383.969,173.002,40.299,157.731
C03183=1048.327,343.402,383.932,173.006,40.303,157.732
C03184=1048.335,343.649,383.896,173.012,40.307,157.733
C03185=1048.342,343.897,383.859,173.016,40.311,157.734
C03186=1048.349,344.143,383.822,173.021,40.315,157.735
C03187=1048.356,344.391,383.786,173.025,40.319,157.736
C03188=1048.363,344.638,383.749,173.031,40.323,157.738
C03189=1048.370,344.885,383.712,173.035,40.327,157.739
C03190=1048.377,345.132,383.675,173.040,40.331,157.740
C03191=1048.385,345.379,383.638,173.044,40.336,157.741
C03192=1048.392,345.627,383.602,173.049,40.339,157.742
C03193=1048.399,345.874,383.565,173.054,40.344,157.743
C03194=1048.406,346.121,383.528,173.059,40.348,157.745
C03195=1048.413,346.369,383.492,173.063,40.352,157.746
C03196=1048.421,346.616,383.454,173.068,40.356,157.747
C03197=1048.429,346.916,383.410,173.074,40.361,157.748
C03198=1048.438,347.216,383.364,173.079,40.366,157.750
C03199=1048.447,347.516,383.320,173.086,40.371,157.751
C03200=1048.456,347.816,383.274,173.091,40.376,157.753
C03201=1048.462,348.064,383.238,173.097,40.380,157.754
C03202=1048.470,348.311,383.201,173.101,40.385,157.755
C03203=1048.478,348.558,383.163,173.106,40.389,157.756
C03204=1048.485,348.805,383.126,173.111,40.393,157.758
C03205=1048.493,349.052,383.089,173.116,40.397,157.759
C03206=1048.500,349.299,383.052,173.121,40.401,157.760
C03207=1048.507,349.547,383.014,173.125,40.405,157.761
C03208=1048.515,349.793,382.977,173.131,40.410,157.762
C03209=1048.521,350.040,382.941,173.135,40.414,157.763
C03210=1048.529,350.288,382.904,173.140,40.418,157.765
C03211=1048.536,350.535,382.866,173.145,40.422,157.766
C03212=1048.543,350.782,382.828,173.150,40.427,157.767
C03213=1048.550,351.029,382.791,173.155,40.431,157.768
C03214=1048.558,351.276,382.754,173.159,40.436,157.770
C03215=1048.566,351.523,382.716,173.165,40.440,157.771
C03216=1048.573,351.770,382.679,173.170,40.444,157.772
C03217=1048.580,352.017,382.641,173.174,40.448,157.773
C03218=1048.587,352.264,382.604,173.180,40.453,157.775
C03219=1048.595,352.511,382.566,173.185,40.457,157.776
C03220=1048.602,352.759,382.529,173.189,40.462,157.777
C03221=1048.609,353.006,382.491,173.195,40.466,157.778
C03222=1048.617,353.252,382.453,173.200,40.470,157.780
C03223=1048.624,353.499,382.416,173.204,40.474,157.781
C03224=1048.631,353.746,382.378,173.210,40.479,157.782
C03225=1048.638,353.994,382.340,173.215,40.483,157.783
C03226=1048.646,354.241,382.303,173.219,40.488,157.785
C03227=1048.653,354.487,382.265,173.225,40.493,157.786
C03228=1048.661,354.735,382.227,173.230,40.497,157.787
C03229=1048.668,354.982,382.189,173.236,40.501,157.788
C03230=1048.675,355.229,382.152,173.240,40.506,157.790
C03231=1048.683,355.476,382.114,173.245,40.510,157.791
C03232=1048.690,355.723,382.076,173.251,40.514,157.792
C03233=1048.698,355.970,382.038,173.255,40.519,157.794
C03234=1048.705,356.217,382.000,173.260,40.523,157.795
C03235=1048.713,356.465,381.962,173.266,40.528,157.796
C03236=1048.720,356.711,381.924,173.271,40.532,157.798
C03237=1048.728,356.958,381.887,173.277,40.537,157.799
C03238=1048.735,357.205,381.848,173.281,40.541,157.800
C03239=1048.743,357.452,381.811,173.287,40.546,157.802
C03240=1048.751,357.699,381.772,173.292,40.550,157.803
C03241=1048.758,357.946,381.735,173.297,40.555,157.804
C03242=1048.765,358.193,381.696,173.302,40.560,157.805
C03243=1048.772,358.439,381.658,173.307,40.564,157.807
C03244=1048.780,358.687,381.620,173.313,40.569,157.808
C03245=1048.788,358.934,381.581,173.318,40.573,157.809
C03246=1048.795,359.180,381.543,173.323,40.578,157.811
C03247=1048.802,359.427,381.504,173.328,40.583,157.812
C03248=1048.810,359.675,381.466,173.333,40.587,157.813
C03249=1048.817,359.922,381.428,173.339,40.592,157.815
C03250=1048.825,360.168,381.390,173.344,40.596,157.816
C03251=1048.832,360.415,381.351,173.350,40.601,157.817
C03252=1048.840,360.662,381.313,173.355,40.606,157.819
C03253=1048.849,360.967,381.265,173.361,40.612,157.821
C03254=1048.858,361.273,381.218,173.368,40.617,157.822
C03255=1048.868,361.580,381.170,173.375,40.623,157.824
C03256=1048.877,361.885,381.123,173.382,40.629,157.826
C03257=1048.885,362.132,381.084,173.387,40.634,157.827
C03258=1048.892,362.379,381.046,173.393,40.638,157.828
C03259=1048.900,362.625,381.007,173.397,40.643,157.830
C03260=1048.907,362.873,380.968,173.403,40.648,157.831
C03261=1048.915,363.119,380.930,173.408,40.653,157.833
C03262=1048.923,363.366,380.890,173.414,40.657,157.834
C03263=1048.930,363.613,380.852,173.419,40.663,157.835
C03264=1048.938,363.860,380.813,173.425,40.667,157.837
C03265=1048.945,364.107,380.774,173.430,40.672,157.838
C03266=1048.952,364.353,380.735,173.436,40.677,157.840
C03267=1048.960,364.600,380.696,173.441,40.682,157.841
C03268=1048.967,364.847,380.657,173.447,40.687,157.843
C03269=1048.975,365.094,380.619,173.452,40.692,157.844
C03270=1048.982,365.340,380.579,173.458,40.696,157.845
C03271=1048.991,365.587,380.541,173.464,40.702,157.847
C03272=1048.998,365.834,380.501,173.469,40.706,157.848
C03273=1049.006,366.081,380.462,173.474,40.711,157.850
C03274=1049.013,366.328,380.424,173.479,40.716,157.851
C03275=1049.020,366.575,380.384,173.485,40.721,157.853
C03276=1049.029,366.822,380.345,173.490,40.726,157.854
C03277=1049.036,367.068,380.305,173.496,40.731,157.856
C03278=1049.044,367.315,380.267,173.502,40.736,157.857
C03279=1049.051,367.561,380.227,173.507,40.741,157.859
C03280=1049.059,367.808,380.188,173.514,40.746,157.860
C03281=1049.067,368.056,380.149,173.520,40.751,157.861
C03282=1049.074,368.302,380.109,173.525,40.756,157.863
C03283=1049.082,368.548,380.070,173.531,40.761,157.864
C03284=1049.090,368.796,380.031,173.537,40.766,157.866
C03285=1049.098,369.042,379.992,173.542,40.771,157.867
C03286=1049.105,369.289,379.952,173.548,40.776,157.869
C03287=1049.114,369.536,379.913,173.553,40.781,157.870
C03288=1049.121,369.783,379.873,173.559,40.786,157.872
C03289=1049.128,370.029,379.834,173.565,40.791,157.873
C03290=1049.137,370.276,379.794,173.570,40.796,157.875
C03291=1049.145,370.523,379.755,173.576,40.801,157.876
C03292=1049.153,370.769,379.715,173.582,40.807,157.878
C03293=1049.160,371.016,379.676,173.588,40.812,157.879
C03294=1049.168,371.263,379.636,173.594,40.817,157.881
C03295=1049.176,371.509,379.597,173.600,40.822,157.882
C03296=1049.184,371.756,379.557,173.605,40.827,157.884
C03297=1049.191,372.003,379.517,173.611,40.832,157.886
C03298=1049.199,372.249,379.477,173.617,40.837,157.887
C03299=1049.207,372.496,379.437,173.622,40.843,157.889
C03300=1049.214,372.743,379.397,173.628,40.848,157.890
C03301=1049.222,372.990,379.357,173.635,40.854,157.892
C03302=1049.230,373.236,379.317,173.641,40.859,157.894
C03303=1049.237,373.482,379.277,173.647,40.864,157.895
C03304=1049.245,373.729,379.237,173.652,40.869,157.897
C03305=1049.253,373.976,379.197,173.658,40.875,157.898
C03306=1049.261,374.222,379.158,173.665,40.880,157.900
C03307=1049.269,374.469,379.117,173.671,40.885,157.901
C03308=1049.277,374.716,379.077,173.676,40.891,157.903
C03309=1049.287,375.041,379.024,173.684,40.898,157.905
C03310=1049.297,375.365,378.972,173.692,40.905,157.907
C03311=1049.308,375.690,378.919,173.700,40.912,157.909
C03312=1049.318,376.015,378.865,173.708,40.919,157.911
C03313=1049.326,376.261,378.825,173.714,40.925,157.913
C03314=1049.334,376.508,378.785,173.720,40.930,157.915
C03315=1049.342,376.754,378.744,173.726,40.935,157.916
C03316=1049.349,377.001,378.704,173.732,40.941,157.918
C03317=1049.357,377.248,378.664,173.739,40.946,157.920
C03318=1049.365,377.494,378.623,173.745,40.952,157.921
C03319=1049.373,377.741,378.583,173.750,40.957,157.923
C03320=1049.382,377.987,378.543,173.757,40.963,157.925
C03321=1049.390,378.233,378.502,173.763,40.968,157.926
C03322=1049.398,378.481,378.462,173.769,40.974,157.928
C03323=1049.406,378.727,378.421,173.776,40.979,157.930
C03324=1049.414,378.973,378.381,173.782,40.984,157.931
C03325=1049.422,379.219,378.340,173.788,40.990,157.933
C03326=1049.430,379.466,378.300,173.795,40.996,157.935
C03327=1049.439,379.713,378.259,173.800,41.002,157.936
C03328=1049.446,379.960,378.218,173.806,41.007,157.938
C03329=1049.454,380.206,378.177,173.813,41.012,157.940
C03330=1049.462,380.452,378.136,173.819,41.018,157.941
C03331=1049.470,380.698,378.095,173.825,41.024,157.943
C03332=1049.478,380.945,378.054,173.832,41.030,157.945
C03333=1049.486,381.192,378.013,173.838,41.035,157.947
C03334=1049.494,381.438,377.973,173.845,41.041,157.948
C03335=1049.501,381.685,377.931,173.851,41.047,157.950
C03336=1049.510,381.931,377.891,173.857,41.053,157.952
C03337=1049.518,382.177,377.849,173.864,41.059,157.954
C03338=1049.526,382.424,377.808,173.870,41.065,157.955
C03339=1049.534,382.670,377.767,173.877,41.070,157.957
C03340=1049.542,382.916,377.727,173.883,41.076,157.959
C03341=1049.550,383.163,377.684,173.890,41.082,157.961
C03342=1049.558,383.409,377.644,173.896,41.088,157.962
C03343=1049.566,383.655,377.602,173.903,41.093,157.964
C03344=1049.574,383.902,377.561,173.909,41.099,157.966
C03345=1049.582,384.149,377.520,173.916,41.105,157.968
C03346=1049.591,384.394,377.479,173.922,41.111,157.970
C03347=1049.598,384.642,377.437,173.929,41.117,157.971
C03348=1049.607,384.887,377.396,173.935,41.123,157.973
C03349=1049.615,385.134,377.355,173.942,41.129,157.975
C03350=1049.623,385.380,377.313,173.948,41.135,157.977
C03351=1049.632,385.627,377.271,173.955,41.141,157.979
C03352=1049.640,385.873,377.230,173.961,41.147,157.981
C03353=1049.648,386.120,377.188,173.968,41.152,157.982
C03354=1049.657,386.365,377.147,173.975,41.159,157.984
C03355=1049.664,386.612,377.105,173.981,41.165,157.986
C03356=1049.673,386.858,377.064,173.988,41.170,157.988
C03357=1049.682,387.105,377.022,173.994,41.177,157.990
C03358=1049.689,387.350,376.980,174.002,41.183,157.992
C03359=1049.698,387.597,376.938,174.009,41.188,157.993
C03360=1049.707,387.844,376.897,174.015,41.195,157.995
C03361=1049.714,388.090,376.855,174.022,41.201,157.997
C03362=1049.723,388.336,376.814,174.029,41.207,157.999
C03363=1049.731,388.582,376.772,174.035,41.213,158.001
C03364=1049.740,388.828,376.730,174.042,41.219,158.003
C03365=1049.752,389.186,376.669,174.053,41.228,158.006
C03366=1049.764,389.543,376.608,174.063,41.237,158.008
C03367=1049.776,389.901,376.547,174.072,41.246,158.011
C03368=1049.788,390.258,376.486,174.082,41.256,158.014
C03369=1049.796,390.504,376.443,174.089,41.262,158.016
C03370=1049.805,390.751,376.401,174.096,41.268,158.018
C03371=1049.814,390.998,376.359,174.103,41.275,158.020
C03372=1049.822,391.243,376.316,174.110,41.281,158.022
C03373=1049.830,391.489,376.275,174.117,41.287,158.024
C03374=1049.839,391.736,376.232,174.125,41.293,158.026
C03375=1049.847,391.982,376.189,174.131,41.300,158.028
C03376=1049.856,392.228,376.148,174.138,41.306,158.030
C03377=1049.864,392.474,376.105,174.145,41.313,158.032
C03378=1049.872,392.720,376.063,174.153,41.319,158.034
C03379=1049.881,392.966,376.020,174.160,41.325,158.036
C03380=1049.890,393.213,375.978,174.166,41.332,158.038
C03381=1049.898,393.459,375.935,174.174,41.338,158.040
C03382=1049.907,393.705,375.892,174.181,41.345,158.042
C03383=1049.915,393.952,375.850,174.188,41.352,158.044
C03384=1049.923,394.197,375.807,174.195,41.358,158.046
C03385=1049.931,394.443,375.764,174.203,41.364,158.048
C03386=1049.940,394.689,375.722,174.210,41.371,158.050
C03387=1049.949,394.935,375.678,174.218,41.378,158.052
C03388=1049.957,395.181,375.636,174.224,41.384,158.054
C03389=1049.966,395.427,375.593,174.231,41.391,158.056
C03390=1049.974,395.674,375.550,174.239,41.398,158.058
C03391=1049.983,395.920,375.507,174.246,41.404,158.060
C03392=1049.992,396.165,375.465,174.254,41.411,158.062
C03393=1050.000,396.411,375.422,174.261,41.418,158.065
C03394=1050.009,396.657,375.379,174.269,41.424,158.067
C03395=1050.018,396.904,375.335,174.276,41.431,158.069
C03396=1050.027,397.150,375.292,174.283,41.437,158.071
C03397=1050.035,397.396,375.248,174.291,41.445,158.073
C03398=1050.044,397.642,375.205,174.298,41.451,158.075
C03399=1050.052,397.888,375.162,174.306,41.458,158.077
C03400=1050.061,398.134,375.119,174.313,41.465,158.079
C03401=1050.069,398.380,375.076,174.321,41.472,158.082
C03402=1050.077,398.626,375.032,174.328,41.478,158.084
C03403=1050.086,398.872,374.989,174.336,41.485,158.086
C03404=1050.095,399.118,374.945,174.343,41.492,158.088
C03405=1050.104,399.364,374.902,174.351,41.499,158.090
C03406=1050.112,399.610,374.859,174.358,41.506,158.092
C03407=1050.122,399.856,374.815,174.366,41.513,158.095
C03408=1050.130,400.102,374.772,174.374,41.520,158.097
C03409=1050.139,400.348,374.728,174.381,41.527,158.099
C03410=1050.148,400.594,374.685,174.390,41.534,158.101
C03411=1050.157,400.840,374.641,174.397,41.541,158.104
C03412=1050.166,401.086,374.597,174.405,41.548,158.106
C03413=1050.174,401.332,374.553,174.413,41.555,158.108
C03414=1050.183,401.578,374.509,174.420,41.562,158.110
C03415=1050.192,401.824,374.465,174.428,41.569,158.113
C03416=1050.201,402.069,374.421,174.436,41.577,158.115
C03417=1050.210,402.316,374.378,174.444,41.583,158.117
C03418=1050.218,402.562,374.334,174.452,41.591,158.119
C03419=1050.228,402.808,374.290,174.459,41.598,158.122
C03420=1050.237,403.053,374.246,174.467,41.605,158.124
C03421=1050.250,403.430,374.179,174.479,41.616,158.127
C03422=1050.263,403.805,374.111,174.491,41.627,158.131
C03423=1050.277,404.182,374.043,174.504,41.638,158.135
C03424=1050.290,404.558,373.976,174.516,41.650,158.138
C03425=1050.300,404.804,373.932,174.525,41.656,158.140
C03426=1050.309,405.050,373.886,174.532,41.664,158.143
C03427=1050.317,405.295,373.842,174.540,41.672,158.145
C03428=1050.326,405.541,373.798,174.549,41.679,158.148
C03429=1050.335,405.786,373.753,174.557,41.686,158.150
C03430=1050.344,406.033,373.708,174.565,41.694,158.152
C03431=1050.353,406.279,373.664,174.574,41.702,158.155
C03432=1050.362,406.525,373.619,174.581,41.709,158.157
C03433=1050.371,406.770,373.575,174.589,41.716,158.160
C03434=1050.380,407.016,373.530,174.598,41.724,158.162
C03435=1050.390,407.262,373.486,174.606,41.731,158.165
C03436=1050.399,407.508,373.440,174.615,41.739,158.167
C03437=1050.407,407.753,373.395,174.623,41.746,158.169
C03438=1050.416,407.999,373.351,174.632,41.754,158.172
C03439=1050.425,408.245,373.306,174.640,41.762,158.174
C03440=1050.435,408.490,373.261,174.648,41.770,158.177
C03441=1050.444,408.737,373.216,174.657,41.777,158.179
C03442=1050.453,408.982,373.171,174.664,41.785,158.182
C03443=1050.462,409.228,373.126,174.674,41.793,158.184
C03444=1050.471,409.474,373.080,174.682,41.800,158.187
C03445=1050.481,409.720,373.036,174.691,41.808,158.190
C03446=1050.490,409.965,372.990,174.700,41.816,158.192
C03447=1050.500,410.211,372.945,174.707,41.823,158.194
C03448=1050.509,410.457,372.900,174.717,41.831,158.197
C03449=1050.518,410.702,372.855,174.725,41.840,158.200
C03450=1050.527,410.948,372.810,174.734,41.847,158.202
C03451=1050.536,411.194,372.764,174.743,41.855,158.205
C03452=1050.546,411.439,372.720,174.751,41.863,158.207
C03453=1050.555,411.685,372.674,174.760,41.871,158.210
C03454=1050.564,411.931,372.629,174.769,41.879,158.213
C03455=1050.575,412.177,372.583,174.777,41.887,158.215
C03456=1050.584,412.422,372.537,174.786,41.895,158.218
C03457=1050.593,412.668,372.493,174.795,41.903,158.220
C03458=1050.603,412.913,372.446,174.805,41.911,158.223
C03459=1050.612,413.160,372.401,174.813,41.919,158.226
C03460=1050.622,413.405,372.354,174.822,41.927,158.229
C03461=1050.630,413.651,372.309,174.831,41.935,158.231
C03462=1050.640,413.896,372.263,174.840,41.943,158.234
C03463=1050.649,414.143,372.217,174.849,41.952,158.237
C03464=1050.659,414.388,372.171,174.858,41.960,158.239
C03465=1050.669,414.633,372.125,174.867,41.968,158.242
C03466=1050.678,414.878,372.080,174.876,41.976,158.245
C03467=1050.688,415.124,372.034,174.886,41.985,158.248
C03468=1050.697,415.370,371.987,174.895,41.992,158.250
C03469=1050.707,415.615,371.941,174.903,42.001,158.253
C03470=1050.716,415.861,371.895,174.913,42.010,158.256
C03471=1050.725,416.106,371.849,174.922,42.017,158.258
C03472=1050.735,416.352,371.802,174.931,42.026,158.261
C03473=1050.744,416.597,371.756,174.941,42.034,158.264
C03474=1050.754,416.843,371.710,174.950,42.043,158.267
C03475=1050.764,417.088,371.663,174.960,42.051,158.270
C03476=1050.773,417.334,371.617,174.969,42.060,158.273
C03477=1050.788,417.717,371.545,174.983,42.073,158.277
C03478=1050.804,418.099,371.472,174.999,42.087,158.282
C03479=1050.819,418.482,371.400,175.013,42.100,158.286
C03480=1050.834,418.864,371.327,175.029,42.113,158.291
C03481=1050.844,419.110,371.280,175.038,42.122,158.293
C03482=1050.854,419.355,371.233,175.048,42.131,158.296
C03483=1050.863,419.601,371.187,175.057,42.139,158.299
C03484=1050.873,419.846,371.139,175.067,42.148,158.302
C03485=1050.883,420.092,371.092,175.078,42.157,158.305
C03486=1050.892,420.337,371.046,175.087,42.165,158.308
C03487=1050.903,420.582,370.998,175.097,42.174,158.311
C03488=1050.912,420.828,370.951,175.106,42.183,158.314
C03489=1050.922,421.073,370.903,175.116,42.192,158.317
C03490=1050.932,421.318,370.857,175.127,42.201,158.320
C03491=1050.942,421.563,370.810,175.136,42.210,158.323
C03492=1050.951,421.809,370.762,175.146,42.219,158.326
C03493=1050.961,422.054,370.715,175.156,42.228,158.329
C03494=1050.972,422.300,370.668,175.167,42.237,158.332
C03495=1050.981,422.545,370.620,175.176,42.246,158.335
C03496=1050.991,422.790,370.573,175.186,42.255,158.338
C03497=1051.002,423.035,370.525,175.197,42.264,158.342
C03498=1051.012,423.280,370.478,175.207,42.273,158.345
C03499=1051.021,423.526,370.430,175.217,42.282,158.348
C03500=1051.032,423.771,370.383,175.227,42.291,158.351
C03501=1051.042,424.016,370.335,175.238,42.300,158.354
C03502=1051.052,424.262,370.287,175.248,42.310,158.357
C03503=1051.062,424.507,370.240,175.259,42.319,158.360
C03504=1051.072,424.751,370.192,175.269,42.328,158.364
C03505=1051.082,424.997,370.144,175.280,42.337,158.367
C03506=1051.093,425.242,370.096,175.290,42.346,158.370
C03507=1051.103,425.488,370.048,175.300,42.356,158.373
C03508=1051.113,425.733,370.000,175.311,42.366,158.376
C03509=1051.123,425.977,369.952,175.322,42.375,158.380
C03510=1051.133,426.224,369.904,175.332,42.384,158.383
C03511=1051.144,426.468,369.856,175.343,42.393,158.386
C03512=1051.154,426.713,369.807,175.354,42.403,158.389
C03513=1051.164,426.958,369.759,175.364,42.412,158.393
C03514=1051.174,427.204,369.710,175.375,42.422,158.396
C03515=1051.184,427.449,369.662,175.386,42.432,158.399
C03516=1051.195,427.693,369.614,175.397,42.441,158.403
C03517=1051.205,427.939,369.565,175.407,42.451,158.406
C03518=1051.215,428.184,369.517,175.418,42.461,158.409
C03519=1051.226,428.429,369.468,175.430,42.470,158.413
C03520=1051.236,428.674,369.420,175.441,42.480,158.416
C03521=1051.247,428.919,369.371,175.451,42.490,158.420
C03522=1051.257,429.164,369.322,175.462,42.500,158.423
C03523=1051.268,429.409,369.274,175.473,42.509,158.426
C03524=1051.278,429.654,369.225,175.485,42.519,158.430
C03525=1051.288,429.899,369.176,175.496,42.529,158.433
C03526=1051.298,430.144,369.127,175.507,42.539,158.437
C03527=1051.309,430.389,369.078,175.519,42.549,158.440
C03528=1051.320,430.633,369.029,175.530,42.559,158.444
C03529=1051.330,430.879,368.980,175.541,42.568,158.447
C03530=1051.341,431.124,368.931,175.553,42.579,158.451
C03531=1051.351,431.369,368.881,175.564,42.589,158.454
C03532=1051.362,431.613,368.832,175.576,42.599,158.458
C03533=1051.377,431.952,368.764,175.592,42.613,158.463
C03534=1051.391,432.290,368.696,175.607,42.627,158.468
C03535=1051.406,432.628,368.627,175.623,42.641,158.473
C03536=1051.421,432.966,368.560,175.640,42.655,158.478
C03537=1051.432,433.211,368.509,175.651,42.665,158.481
C03538=1051.442,433.456,368.460,175.664,42.676,158.485
C03539=1051.453,433.701,368.410,175.675,42.686,158.489
C03540=1051.464,433.946,368.361,175.687,42.697,158.493
C03541=1051.475,434.190,368.310,175.699,42.707,158.496
C03542=1051.485,434.435,368.261,175.711,42.717,158.500
C03543=1051.497,434.680,368.212,175.723,42.728,158.504
C03544=1051.508,434.924,368.161,175.735,42.738,158.507
C03545=1051.518,435.170,368.112,175.747,42.748,158.511
C03546=1051.529,435.414,368.061,175.759,42.759,158.515
C03547=1051.540,435.658,368.011,175.772,42.769,158.519
C03548=1051.551,435.903,367.961,175.784,42.780,158.522
C03549=1051.562,436.148,367.911,175.796,42.791,158.526
C03550=1051.573,436.393,367.860,175.809,42.802,158.530
C03551=1051.584,436.637,367.810,175.820,42.812,158.534
C03552=1051.595,436.882,367.760,175.833,42.823,158.538
C03553=1051.606,437.126,367.709,175.846,42.833,158.542
C03554=1051.617,437.371,367.659,175.858,42.845,158.546
C03555=1051.629,437.616,367.608,175.871,42.855,158.550
C03556=1051.640,437.860,367.558,175.883,42.866,158.554
C03557=1051.651,438.105,367.508,175.896,42.877,158.558
C03558=1051.662,438.350,367.457,175.909,42.888,158.562
C03559=1051.674,438.594,367.406,175.921,42.899,158.566
C03560=1051.685,438.838,367.356,175.934,42.910,158.570
C03561=1051.695,439.084,367.304,175.948,42.921,158.574
C03562=1051.707,439.327,367.253,175.961,42.932,158.578
C03563=1051.719,439.572,367.202,175.973,42.943,158.582
C03564=1051.730,439.816,367.152,175.986,42.955,158.586
C03565=1051.742,440.061,367.100,176.000,42.966,158.590
C03566=1051.752,440.306,367.049,176.013,42.977,158.594
C03567=1051.764,440.550,366.998,176.026,42.988,158.598
C03568=1051.775,440.794,366.947,176.039,42.999,158.603
C03569=1051.787,441.038,366.896,176.053,43.011,158.607
C03570=1051.798,441.283,366.844,176.066,43.022,158.611
C03571=1051.809,441.527,366.793,176.080,43.033,158.615
C03572=1051.821,441.771,366.741,176.093,43.045,158.619
C03573=1051.833,442.016,366.690,176.106,43.056,158.623
C03574=1051.844,442.261,366.638,176.120,43.068,158.628
C03575=1051.855,442.505,366.587,176.133,43.079,158.632
C03576=1051.868,442.749,366.535,176.147,43.091,158.636
C03577=1051.879,442.993,366.483,176.160,43.102,158.641
C03578=1051.891,443.238,366.431,176.175,43.114,158.645
C03579=1051.902,443.482,366.378,176.189,43.126,158.649
C03580=1051.913,443.726,366.327,176.202,43.138,158.654
C03581=1051.926,443.970,366.275,176.216,43.149,158.658
C03582=1051.937,444.214,366.223,176.231,43.161,158.663
C03583=1051.949,444.458,366.171,176.244,43.173,158.667
C03584=1051.960,444.703,366.118,176.258,43.185,158.672
C03585=1051.976,445.014,366.052,176.276,43.200,158.677
C03586=1051.991,445.325,365.985,176.295,43.215,158.683
C03587=1052.007,445.635,365.919,176.313,43.230,158.689
C03588=1052.022,445.947,365.852,176.332,43.246,158.695
C03589=1052.040,446.322,365.771,176.354,43.264,158.702
C03590=1052.061,446.699,365.691,176.376,43.282,158.709
C03591=1052.083,447.077,365.612,176.399,43.300,158.716
C03592=1052.107,447.456,365.535,176.422,43.318,158.722
C03593=1052.123,447.699,365.486,176.437,43.329,158.727
C03594=1052.140,447.943,365.438,176.452,43.340,158.731
C03595=1052.158,448.188,365.390,176.467,43.350,158.735
C03596=1052.176,448.433,365.342,176.482,43.361,158.740
C03597=1052.195,448.678,365.295,176.497,43.371,158.744
C03598=1052.215,448.922,365.249,176.513,43.382,158.748
C03599=1052.237,449.167,365.202,176.528,43.392,158.752
C03600=1052.258,449.412,365.157,176.543,43.402,158.756
C03601=1052.280,449.658,365.112,176.559,43.412,158.760
C03602=1052.304,449.903,365.068,176.575,43.422,158.765
C03603=1052.327,450.147,365.024,176.591,43.431,158.769
C03604=1052.351,450.393,364.982,176.606,43.441,158.773
C03605=1052.034,450.417,364.686,176.605,43.536,158.800
C03606=1052.010,450.172,364.728,176.589,43.527,158.796
C03607=1051.985,449.927,364.772,176.574,43.517,158.792
C03608=1051.963,449.682,364.816,176.558,43.508,158.788
C03609=1051.940,449.436,364.861,176.543,43.498,158.784
C03610=1051.919,449.191,364.906,176.527,43.489,158.780
C03611=1051.897,448.946,364.952,176.512,43.479,158.776
C03612=1051.878,448.701,364.998,176.497,43.468,158.771
C03613=1051.858,448.456,365.045,176.481,43.458,158.767
C03614=1051.839,448.212,365.093,176.466,43.447,158.763
C03615=1051.821,447.967,365.141,176.450,43.437,158.759
C03616=1051.804,447.723,365.189,176.435,43.426,158.754
C03617=1051.788,447.480,365.238,176.420,43.415,158.750
C03618=1051.764,447.120,365.312,176.399,43.398,158.743
C03619=1051.743,446.760,365.386,176.377,43.381,158.737
C03620=1051.724,446.401,365.462,176.355,43.364,158.730
C03621=1051.705,446.045,365.538,176.334,43.347,158.723
C03622=1051.693,445.801,365.591,176.319,43.335,158.719
C03623=1051.681,445.557,365.643,176.305,43.323,158.714
C03624=1051.670,445.313,365.696,176.290,43.311,158.710
C03625=1051.657,445.069,365.748,176.276,43.299,158.705
C03626=1051.645,444.825,365.800,176.261,43.288,158.701
C03627=1051.634,444.581,365.853,176.247,43.276,158.696
C03628=1051.621,444.336,365.905,176.233,43.264,158.692
C03629=1051.610,444.092,365.956,176.219,43.252,158.687
C03630=1051.598,443.848,366.009,176.205,43.240,158.683
C03631=1051.586,443.604,366.060,176.190,43.229,158.679
C03632=1051.575,443.359,366.113,176.177,43.217,158.674
C03633=1051.563,443.115,366.165,176.163,43.206,158.670
C03634=1051.551,442.871,366.217,176.150,43.194,158.666
C03635=1051.540,442.626,366.269,176.135,43.182,158.661
C03636=1051.528,442.382,366.320,176.121,43.171,158.657
C03637=1051.516,442.139,366.372,176.108,43.160,158.653
C03638=1051.505,441.894,366.424,176.094,43.148,158.648
C03639=1051.493,441.649,366.475,176.081,43.137,158.644
C03640=1051.481,441.405,366.527,176.067,43.125,158.640
